KUKA KRL program: EPS_2_25716_MHDR07_A_20250926070400.src

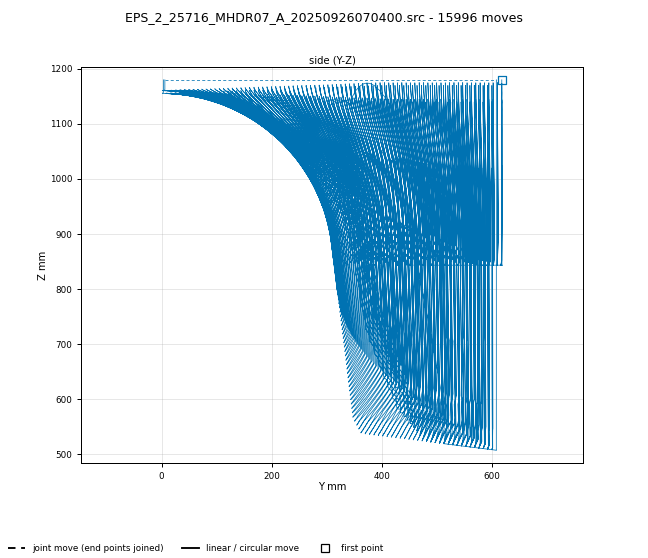
[picture p0: tool path of EPS_2_25716_MHDR07_A_20250926070400.src, 15996 of 15998 moves have a stored position in this frame; points joined in program order, loops and branches not executed]
&ACCESS RVP
&REL 4
&COMMENT QRS 19112012
&PARAM EDITMASK = *
DEF PART()
EXT BAS (BAS_COMMAND :IN,REAL :IN )
INT I
BAS (#INITMOV,0 )

;KUKA QRS Post kuka4.cps  Date:22-06-2017 !

File_ID=2856

QRS_PRE_INIT()

;Init var - Until changes are made in qrs_pre_init
Outlet_Square_prg=0
Inlet_1_Square_prg=0
Inlet_2_Square_prg=0
Inlet_3_Square_prg=0
Inlet_4_Square_prg=0
Inlet_5_Square_prg=0

Outlet_1={X 0.000, Y 400.000, Z 865.000, B 0.000, E1 0.000 }
Inlet_1={X 0.000, Y 425.000, Z 873.500, B 0.000, E1 180.000 }
Inlet_2={X 0.000, Y 495.250, Z 870.500, B 0.000, E1 270.000 }
Outlet_1_type=610
Inlet_1_type=533
Inlet_2_type=299
;QRS#1=Sidecore dimensions
;QRS#2=600-24" Concrete
;QRS#3=525-21" Concrete
;QRS#4=300-12" PVC SDR 35
;QRS#5=
;QRS#6=
;QRS#7=
;QRS#8=
;QRS#9=S306-34L
;QRS#10=S306-32
;QRS#11=16M PSX
;QRS#12=
;QRS#13=
;QRS#14=
;QRS#15=
;QRS#16=1220x127x1524 5'
;QRS#17=EPS Height
;QRS#18=1170
;QRS#19=*
;QRS#20= UPDATED VERSION 22-06-2017
;QRS#21=*
Outlet_Square=0450
Inlet_1_Square=0250
Inlet_2_Square=0150
Inlet_3_Square=0
Inlet_4_Square=0
Inlet_5_Square=0
Mill_Square=1
Outlet_Square_Prg=264
Inlet_1_Square_prg=263
Inlet_2_Square_prg=206

QRS_INIT()

$ADVANCE=5

; T1
PTP {E1 171.027,E2 171.027}
PTP {X 0,Y 617.826,A -85,B 0,C 180,E1 171.027,E2 171.027,E3 0,E4 0,E5 0,E6 0}
QRS_SPEED_INIT()
LIN {X 0,Y 617.826,Z 1180,A -85,B 0,C 180,E1 171.027,E2 171.027,E3 0,E4 0,E5 0,E6 0} C_VEL
LIN {X 0,Y 617.826,Z 845.44,A -85,B 0,C 180,E1 171.027,E2 171.027} C_VEL
LIN {X 0,Y 617.859,Z 843.44,A -85,B 0,C 180,E1 171.213,E2 171.213} C_VEL
LIN {X 0,Y 618.034,Z 843.44,A -85,B 0,C 180,E1 171.886,E2 171.886} C_VEL
LIN {X 0,Y 618.05,Z 843.44,A -85,B 0,C 180,E1 176.532,E2 176.532} C_VEL
LIN {X 0,Y 618.064,Z 843.44,A -85,B 0,C 180,E1 181.155,E2 181.155} C_VEL
LIN {X 0,Y 618.028,Z 843.44,A -85,B 0,C 180,E1 185.786,E2 185.786} C_VEL
LIN {X 0,Y 618.013,Z 843.44,A -85,B 0,C 180,E1 190.456,E2 190.456} C_VEL
LIN {X 0,Y 617.976,Z 843.44,A -85,B 0,C 180,E1 195.197,E2 195.197} C_VEL
LIN {X 0,Y 617.964,Z 843.44,A -85,B 0,C 180,E1 200.048,E2 200.048} C_VEL
LIN {X 0,Y 617.483,Z 843.44,A -85,B 0,C 180,E1 202.547,E2 202.547} C_VEL
LIN {X 0,Y 617.935,Z 843.44,A -85,B 0,C 180,E1 205.055,E2 205.055} C_VEL
LIN {X 0,Y 617.441,Z 843.44,A -85,B 0,C 180,E1 207.658,E2 207.658} C_VEL
LIN {X 0,Y 617.905,Z 843.44,A -85,B 0,C 180,E1 210.277,E2 210.277} C_VEL
LIN {X 0,Y 617.354,Z 843.44,A -85,B 0,C 180,E1 213.025,E2 213.025} C_VEL
LIN {X 0,Y 617.825,Z 843.44,A -85,B 0,C 180,E1 215.797,E2 215.797} C_VEL
LIN {X 0,Y 617.582,Z 843.44,A -85,B 0,C 180,E1 218.101,E2 218.101} C_VEL
LIN {X 0,Y 617.557,Z 843.44,A -85,B 0,C 180,E1 218.721,E2 218.721} C_VEL
LIN {X 0,Y 617.766,Z 843.44,A -85,B 0,C 180,E1 221.733,E2 221.733} C_VEL
LIN {X 0,Y 617.884,Z 843.44,A -85,B 0,C 180,E1 225.1,E2 225.1} C_VEL
LIN {X 0,Y 617.46,Z 843.44,A -85,B 0,C 180,E1 228.307,E2 228.307} C_VEL
LIN {X 0,Y 617.801,Z 843.44,A -85,B 0,C 180,E1 231.297,E2 231.297} C_VEL
LIN {X 0,Y 617.974,Z 843.44,A -85,B 0,C 180,E1 236.343,E2 236.343} C_VEL
LIN {X 0,Y 617.89,Z 843.44,A -85,B 0,C 180,E1 236.673,E2 236.673} C_VEL
LIN {X 0,Y 617.186,Z 843.44,A -85,B 0,C 180,E1 236.798,E2 236.798} C_VEL
LIN {X 0,Y 616.586,Z 843.475,A -85,B 0,C 180,E1 236.859,E2 236.859} C_VEL
LIN {X 0,Y 617.403,Z 850.998,A -85,B 0,C 180,E1 237.011,E2 237.011} C_VEL
LIN {X 0,Y 617.541,Z 885.56,A -85,B 0,C 180,E1 237.498,E2 237.498} C_VEL
LIN {X 0,Y 617.519,Z 896.888,A -85,B 0,C 180,E1 237.684,E2 237.684} C_VEL
LIN {X 0,Y 617.646,Z 911.266,A -85,B 0,C 180,E1 237.997,E2 237.997} C_VEL
LIN {X 0,Y 617.537,Z 922.217,A -85,B 0,C 180,E1 238.279,E2 238.279} C_VEL
LIN {X 0,Y 617.686,Z 929.329,A -85,B 0,C 180,E1 238.492,E2 238.492} C_VEL
LIN {X 0,Y 617.775,Z 942.058,A -85,B 0,C 180,E1 238.905,E2 238.905} C_VEL
LIN {X 0,Y 617.615,Z 958.173,A -85,B 0,C 180,E1 239.505,E2 239.505} C_VEL
LIN {X 0,Y 617.795,Z 971.272,A -85,B 0,C 180,E1 240.077,E2 240.077} C_VEL
LIN {X 0,Y 617.796,Z 985.604,A -85,B 0,C 180,E1 240.772,E2 240.772} C_VEL
LIN {X 0,Y 617.752,Z 997.603,A -85,B 0,C 180,E1 241.411,E2 241.411} C_VEL
LIN {X 0,Y 617.841,Z 1012.189,A -85,B 0,C 180,E1 242.286,E2 242.286} C_VEL
LIN {X 0,Y 617.838,Z 1025.624,A -85,B 0,C 180,E1 243.174,E2 243.174} C_VEL
LIN {X 0,Y 617.827,Z 1037.892,A -85,B 0,C 180,E1 244.06,E2 244.06} C_VEL
LIN {X 0,Y 617.82,Z 1049.111,A -85,B 0,C 180,E1 244.94,E2 244.94} C_VEL
LIN {X 0,Y 617.852,Z 1060.219,A -85,B 0,C 180,E1 245.887,E2 245.887} C_VEL
LIN {X 0,Y 617.902,Z 1071.184,A -85,B 0,C 180,E1 246.902,E2 246.902} C_VEL
LIN {X 0,Y 617.832,Z 1081.53,A -85,B 0,C 180,E1 247.935,E2 247.935} C_VEL
LIN {X 0,Y 617.851,Z 1091.52,A -85,B 0,C 180,E1 249.023,E2 249.023} C_VEL
LIN {X 0,Y 617.958,Z 1100.894,A -85,B 0,C 180,E1 250.135,E2 250.135} C_VEL
LIN {X 0,Y 617.805,Z 1109.459,A -85,B 0,C 180,E1 251.226,E2 251.226} C_VEL
LIN {X 0,Y 617.799,Z 1117.796,A -85,B 0,C 180,E1 252.389,E2 252.389} C_VEL
LIN {X 0,Y 617.999,Z 1125.735,A -85,B 0,C 180,E1 253.612,E2 253.612} C_VEL
LIN {X 0,Y 617.806,Z 1132.883,A -85,B 0,C 180,E1 254.799,E2 254.799} C_VEL
LIN {X 0,Y 617.803,Z 1140.813,A -85,B 0,C 180,E1 256.29,E2 256.29} C_VEL
LIN {X 0,Y 617.952,Z 1146.479,A -85,B 0,C 180,E1 257.48,E2 257.48} C_VEL
LIN {X 0,Y 617.728,Z 1152.733,A -85,B 0,C 180,E1 258.951,E2 258.951} C_VEL
LIN {X 0,Y 617.808,Z 1157.627,A -85,B 0,C 180,E1 260.287,E2 260.287} C_VEL
LIN {X 0,Y 617.981,Z 1160.314,A -85,B 0,C 180,E1 261.14,E2 261.14} C_VEL
LIN {X 0,Y 617.86,Z 1162.559,A -85,B 0,C 180,E1 261.884,E2 261.884} C_VEL
LIN {X 0,Y 617.747,Z 1165.107,A -85,B 0,C 180,E1 262.815,E2 262.815} C_VEL
LIN {X 0,Y 617.832,Z 1168.205,A -85,B 0,C 180,E1 264.212,E2 264.212} C_VEL
LIN {X 0,Y 617.977,Z 1169.802,A -85,B 0,C 180,E1 265.142,E2 265.142} C_VEL
LIN {X 0,Y 617.8,Z 1171.279,A -85,B 0,C 180,E1 266.068,E2 266.068} C_VEL
LIN {X 0,Y 617.755,Z 1172.831,A -85,B 0,C 180,E1 267.456,E2 267.456} C_VEL
LIN {X 0,Y 617.996,Z 1173.642,A -85,B 0,C 180,E1 268.845,E2 268.845} C_VEL
LIN {X 0,Y 617.667,Z 1173.732,A -85,B 0,C 180,E1 271.156,E2 271.156} C_VEL
LIN {X 0,Y 617.779,Z 1173.15,A -85,B 0,C 180,E1 272.081,E2 272.081} C_VEL
LIN {X 0,Y 617.843,Z 1171.818,A -85,B 0,C 180,E1 273.469,E2 273.469} C_VEL
LIN {X 0,Y 617.732,Z 1170.658,A -85,B 0,C 180,E1 274.396,E2 274.396} C_VEL
LIN {X 0,Y 617.804,Z 1168.213,A -85,B 0,C 180,E1 275.788,E2 275.788} C_VEL
LIN {X 0,Y 617.987,Z 1166.125,A -85,B 0,C 180,E1 276.716,E2 276.716} C_VEL
LIN {X 0,Y 617.83,Z 1163.821,A -85,B 0,C 180,E1 277.65,E2 277.65} C_VEL
LIN {X 0,Y 617.779,Z 1160.464,A -85,B 0,C 180,E1 278.831,E2 278.831} C_VEL
LIN {X 0,Y 617.962,Z 1156.403,A -85,B 0,C 180,E1 280.049,E2 280.049} C_VEL
LIN {X 0,Y 617.793,Z 1151.563,A -85,B 0,C 180,E1 281.342,E2 281.342} C_VEL
LIN {X 0,Y 617.737,Z 1146.524,A -85,B 0,C 180,E1 282.524,E2 282.524} C_VEL
LIN {X 0,Y 617.97,Z 1139.3,A -85,B 0,C 180,E1 284.003,E2 284.003} C_VEL
LIN {X 0,Y 617.801,Z 1131.858,A -85,B 0,C 180,E1 285.375,E2 285.375} C_VEL
LIN {X 0,Y 617.792,Z 1124.027,A -85,B 0,C 180,E1 286.666,E2 286.666} C_VEL
LIN {X 0,Y 617.957,Z 1116.024,A -85,B 0,C 180,E1 287.859,E2 287.859} C_VEL
LIN {X 0,Y 617.818,Z 1107.948,A -85,B 0,C 180,E1 288.977,E2 288.977} C_VEL
LIN {X 0,Y 617.839,Z 1098.142,A -85,B 0,C 180,E1 290.206,E2 290.206} C_VEL
LIN {X 0,Y 617.953,Z 1088.763,A -85,B 0,C 180,E1 291.283,E2 291.283} C_VEL
LIN {X 0,Y 617.848,Z 1078.488,A -85,B 0,C 180,E1 292.376,E2 292.376} C_VEL
LIN {X 0,Y 617.845,Z 1068.723,A -85,B 0,C 180,E1 293.335,E2 293.335} C_VEL
LIN {X 0,Y 617.863,Z 1057.185,A -85,B 0,C 180,E1 294.376,E2 294.376} C_VEL
LIN {X 0,Y 617.852,Z 1046.139,A -85,B 0,C 180,E1 295.298,E2 295.298} C_VEL
LIN {X 0,Y 617.837,Z 1033.554,A -85,B 0,C 180,E1 296.261,E2 296.261} C_VEL
LIN {X 0,Y 617.822,Z 1022.09,A -85,B 0,C 180,E1 297.07,E2 297.07} C_VEL
LIN {X 0,Y 617.849,Z 1008.689,A -85,B 0,C 180,E1 297.929,E2 297.929} C_VEL
LIN {X 0,Y 617.812,Z 994.844,A -85,B 0,C 180,E1 298.735,E2 298.735} C_VEL
LIN {X 0,Y 617.727,Z 983.672,A -85,B 0,C 180,E1 299.334,E2 299.334} C_VEL
LIN {X 0,Y 617.802,Z 968.456,A -85,B 0,C 180,E1 300.051,E2 300.051} C_VEL
LIN {X 0,Y 617.675,Z 953.097,A -85,B 0,C 180,E1 300.694,E2 300.694} C_VEL
LIN {X 0,Y 617.671,Z 944.829,A -85,B 0,C 180,E1 300.998,E2 300.998} C_VEL
LIN {X 0,Y 617.767,Z 935.829,A -85,B 0,C 180,E1 301.299,E2 301.299} C_VEL
LIN {X 0,Y 617.783,Z 926.098,A -85,B 0,C 180,E1 301.604,E2 301.604} C_VEL
LIN {X 0,Y 617.523,Z 910.516,A -85,B 0,C 180,E1 302.028,E2 302.028} C_VEL
LIN {X 0,Y 617.755,Z 895.124,A -85,B 0,C 180,E1 302.336,E2 302.336} C_VEL
LIN {X 0,Y 617.696,Z 875.17,A -85,B 0,C 180,E1 302.644,E2 302.644} C_VEL
LIN {X 0,Y 617.35,Z 850.291,A -85,B 0,C 180,E1 303.002,E2 303.002} C_VEL
LIN {X 0,Y 616.629,Z 843.44,A -85,B 0,C 180,E1 303.146,E2 303.146} C_VEL
LIN {X 0,Y 617.119,Z 843.44,A -85,B 0,C 180,E1 303.195,E2 303.195} C_VEL
LIN {X 0,Y 617.816,Z 843.44,A -85,B 0,C 180,E1 303.308,E2 303.308} C_VEL
LIN {X 0,Y 618.037,Z 843.44,A -85,B 0,C 180,E1 303.607,E2 303.607} C_VEL
LIN {X 0,Y 617.768,Z 843.44,A -85,B 0,C 180,E1 305.801,E2 305.801} C_VEL
LIN {X 0,Y 617.724,Z 843.44,A -85,B 0,C 180,E1 308.117,E2 308.117} C_VEL
LIN {X 0,Y 617.813,Z 843.44,A -85,B 0,C 180,E1 311.73,E2 311.73} C_VEL
LIN {X 0,Y 617.416,Z 843.44,A -85,B 0,C 180,E1 315.057,E2 315.057} C_VEL
LIN {X 0,Y 617.813,Z 843.44,A -85,B 0,C 180,E1 318.27,E2 318.27} C_VEL
LIN {X 0,Y 617.717,Z 843.44,A -85,B 0,C 180,E1 321.884,E2 321.884} C_VEL
LIN {X 0,Y 617.729,Z 843.44,A -85,B 0,C 180,E1 324.196,E2 324.196} C_VEL
LIN {X 0,Y 617.802,Z 843.44,A -85,B 0,C 180,E1 325.791,E2 325.791} C_VEL
LIN {X 0,Y 617.831,Z 843.44,A -85,B 0,C 180,E1 327.004,E2 327.004} C_VEL
LIN {X 0,Y 618.061,Z 843.44,A -85,B 0,C 180,E1 331.451,E2 331.451} C_VEL
LIN {X 0,Y 617.532,Z 843.44,A -85,B 0,C 180,E1 335.24,E2 335.24} C_VEL
LIN {X 0,Y 617.711,Z 843.44,A -85,B 0,C 180,E1 337.462,E2 337.462} C_VEL
LIN {X 0,Y 617.977,Z 843.44,A -85,B 0,C 180,E1 342.394,E2 342.394} C_VEL
LIN {X 0,Y 617.279,Z 843.44,A -85,B 0,C 180,E1 342.777,E2 342.777} C_VEL
LIN {X 0,Y 616.404,Z 843.44,A -85,B 0,C 180,E1 342.867,E2 342.867} C_VEL
LIN {X 0,Y 617.46,Z 848.376,A -85,B 0,C 180,E1 342.958,E2 342.958} C_VEL
LIN {X 0,Y 617.866,Z 852.602,A -85,B 0,C 180,E1 343.02,E2 343.02} C_VEL
LIN {X 0,Y 617.94,Z 873.653,A -85,B 0,C 180,E1 343.286,E2 343.286} C_VEL
LIN {X 0,Y 617.951,Z 884.015,A -85,B 0,C 180,E1 343.474,E2 343.474} C_VEL
LIN {X 0,Y 617.935,Z 894.426,A -85,B 0,C 180,E1 343.73,E2 343.73} C_VEL
LIN {X 0,Y 618.005,Z 903.309,A -85,B 0,C 180,E1 344,E2 344} C_VEL
LIN {X 0,Y 617.986,Z 911.677,A -85,B 0,C 180,E1 344.297,E2 344.297} C_VEL
LIN {X 0,Y 617.988,Z 918.429,A -85,B 0,C 180,E1 344.571,E2 344.571} C_VEL
LIN {X 0,Y 618.018,Z 926.731,A -85,B 0,C 180,E1 344.953,E2 344.953} C_VEL
LIN {X 0,Y 618.01,Z 935.331,A -85,B 0,C 180,E1 345.401,E2 345.401} C_VEL
LIN {X 0,Y 617.98,Z 945.261,A -85,B 0,C 180,E1 345.997,E2 345.997} C_VEL
LIN {X 0,Y 617.998,Z 952.881,A -85,B 0,C 180,E1 346.518,E2 346.518} C_VEL
LIN {X 0,Y 618.001,Z 959.746,A -85,B 0,C 180,E1 347.037,E2 347.037} C_VEL
LIN {X 0,Y 617.986,Z 966.834,A -85,B 0,C 180,E1 347.629,E2 347.629} C_VEL
LIN {X 0,Y 617.989,Z 974.718,A -85,B 0,C 180,E1 348.367,E2 348.367} C_VEL
LIN {X 0,Y 617.99,Z 980.34,A -85,B 0,C 180,E1 348.956,E2 348.956} C_VEL
LIN {X 0,Y 618.005,Z 985.465,A -85,B 0,C 180,E1 349.544,E2 349.544} C_VEL
LIN {X 0,Y 617.972,Z 991.481,A -85,B 0,C 180,E1 350.309,E2 350.309} C_VEL
LIN {X 0,Y 617.952,Z 996.842,A -85,B 0,C 180,E1 351.072,E2 351.072} C_VEL
LIN {X 0,Y 617.99,Z 1001.905,A -85,B 0,C 180,E1 351.886,E2 351.886} C_VEL
LIN {X 0,Y 617.944,Z 1006.92,A -85,B 0,C 180,E1 352.818,E2 352.818} C_VEL
LIN {X 0,Y 617.915,Z 1010.212,A -85,B 0,C 180,E1 353.516,E2 353.516} C_VEL
LIN {X 0,Y 617.956,Z 1013.094,A -85,B 0,C 180,E1 354.213,E2 354.213} C_VEL
LIN {X 0,Y 617.988,Z 1014.821,A -85,B 0,C 180,E1 354.678,E2 354.678} C_VEL
LIN {X 0,Y 617.913,Z 1017.797,A -85,B 0,C 180,E1 355.605,E2 355.605} C_VEL
LIN {X 0,Y 617.894,Z 1020.135,A -85,B 0,C 180,E1 356.531,E2 356.531} C_VEL
LIN {X 0,Y 617.975,Z 1021.885,A -85,B 0,C 180,E1 357.457,E2 357.457} C_VEL
LIN {X 0,Y 617.978,Z 1022.566,A -85,B 0,C 180,E1 357.92,E2 357.92} C_VEL
LIN {X 0,Y 617.893,Z 1023.509,A -85,B 0,C 180,E1 358.844,E2 358.844} C_VEL
LIN {X 0,Y 617.884,Z 1023.799,A -85,B 0,C 180,E1 359.307,E2 359.307} C_VEL
LIN {X 0,Y 617.958,Z 1023.865,A -85,B 0,C 180,E1 360.231,E2 360.231} C_VEL
LIN {X 0,Y 617.93,Z 1023.435,A -85,B 0,C 180,E1 361.156,E2 361.156} C_VEL
LIN {X 0,Y 617.886,Z 1023.032,A -85,B 0,C 180,E1 361.618,E2 361.618} C_VEL
LIN {X 0,Y 617.897,Z 1021.756,A -85,B 0,C 180,E1 362.543,E2 362.543} C_VEL
LIN {X 0,Y 617.989,Z 1019.915,A -85,B 0,C 180,E1 363.468,E2 363.468} C_VEL
LIN {X 0,Y 617.905,Z 1017.555,A -85,B 0,C 180,E1 364.395,E2 364.395} C_VEL
LIN {X 0,Y 617.893,Z 1014.509,A -85,B 0,C 180,E1 365.323,E2 365.323} C_VEL
LIN {X 0,Y 617.929,Z 1012.766,A -85,B 0,C 180,E1 365.787,E2 365.787} C_VEL
LIN {X 0,Y 617.981,Z 1008.74,A -85,B 0,C 180,E1 366.716,E2 366.716} C_VEL
LIN {X 0,Y 617.924,Z 1004.006,A -85,B 0,C 180,E1 367.649,E2 367.649} C_VEL
LIN {X 0,Y 617.961,Z 998.442,A -85,B 0,C 180,E1 368.595,E2 368.595} C_VEL
LIN {X 0,Y 618.003,Z 993.303,A -85,B 0,C 180,E1 369.355,E2 369.355} C_VEL
LIN {X 0,Y 617.953,Z 987.738,A -85,B 0,C 180,E1 370.089,E2 370.089} C_VEL
LIN {X 0,Y 617.968,Z 982.163,A -85,B 0,C 180,E1 370.75,E2 370.75} C_VEL
LIN {X 0,Y 618.001,Z 975.273,A -85,B 0,C 180,E1 371.485,E2 371.485} C_VEL
LIN {X 0,Y 617.99,Z 967.501,A -85,B 0,C 180,E1 372.223,E2 372.223} C_VEL
LIN {X 0,Y 617.991,Z 960.481,A -85,B 0,C 180,E1 372.815,E2 372.815} C_VEL
LIN {X 0,Y 618.01,Z 953.686,A -85,B 0,C 180,E1 373.334,E2 373.334} C_VEL
LIN {X 0,Y 618.026,Z 946.145,A -85,B 0,C 180,E1 373.853,E2 373.853} C_VEL
LIN {X 0,Y 618.015,Z 936.423,A -85,B 0,C 180,E1 374.449,E2 374.449} C_VEL
LIN {X 0,Y 617.982,Z 927.966,A -85,B 0,C 180,E1 374.898,E2 374.898} C_VEL
LIN {X 0,Y 618.015,Z 919.027,A -85,B 0,C 180,E1 375.312,E2 375.312} C_VEL
LIN {X 0,Y 618.031,Z 910.408,A -85,B 0,C 180,E1 375.66,E2 375.66} C_VEL
LIN {X 0,Y 617.966,Z 901.85,A -85,B 0,C 180,E1 375.959,E2 375.959} C_VEL
LIN {X 0,Y 618.01,Z 891.38,A -85,B 0,C 180,E1 376.262,E2 376.262} C_VEL
LIN {X 0,Y 617.964,Z 880.659,A -85,B 0,C 180,E1 376.501,E2 376.501} C_VEL
LIN {X 0,Y 617.886,Z 871.697,A -85,B 0,C 180,E1 376.653,E2 376.653} C_VEL
LIN {X 0,Y 617.825,Z 844.104,A -85,B 0,C 180,E1 376.992,E2 376.992} C_VEL
LIN {X 0,Y 617.73,Z 843.44,A -85,B 0,C 180,E1 377.012,E2 377.012} C_VEL
LIN {X 0,Y 618.008,Z 843.44,A -85,B 0,C 180,E1 377.344,E2 377.344} C_VEL
LIN {X 0,Y 617.906,Z 843.44,A -85,B 0,C 180,E1 382.53,E2 382.53} C_VEL
LIN {X 0,Y 617.419,Z 843.44,A -85,B 0,C 180,E1 385.077,E2 385.077} C_VEL
LIN {X 0,Y 617.864,Z 843.44,A -85,B 0,C 180,E1 387.637,E2 387.637} C_VEL
LIN {X 0,Y 617.41,Z 843.44,A -85,B 0,C 180,E1 390.304,E2 390.304} C_VEL
LIN {X 0,Y 617.944,Z 843.44,A -85,B 0,C 180,E1 392.989,E2 392.989} C_VEL
LIN {X 0,Y 617.692,Z 843.44,A -85,B 0,C 180,E1 395.806,E2 395.806} C_VEL
LIN {X 0,Y 617.698,Z 843.44,A -85,B 0,C 180,E1 398.114,E2 398.114} C_VEL
LIN {X 0,Y 617.763,Z 843.44,A -85,B 0,C 180,E1 401.734,E2 401.734} C_VEL
LIN {X 0,Y 617.403,Z 843.44,A -85,B 0,C 180,E1 405.055,E2 405.055} C_VEL
LIN {X 0,Y 617.813,Z 843.44,A -85,B 0,C 180,E1 408.27,E2 408.27} C_VEL
LIN {X 0,Y 617.726,Z 843.44,A -85,B 0,C 180,E1 411.882,E2 411.882} C_VEL
LIN {X 0,Y 617.761,Z 843.44,A -85,B 0,C 180,E1 414.198,E2 414.198} C_VEL
LIN {X 0,Y 617.859,Z 843.44,A -85,B 0,C 180,E1 415.783,E2 415.783} C_VEL
LIN {X 0,Y 617.919,Z 843.44,A -85,B 0,C 180,E1 417.01,E2 417.01} C_VEL
LIN {X 0,Y 618.055,Z 843.44,A -85,B 0,C 180,E1 420.692,E2 420.692} C_VEL
LIN {X 0,Y 616.955,Z 843.44,A -85,B 0,C 180,E1 420.924,E2 420.924} C_VEL
LIN {X 0,Y 617.601,Z 885.711,A -85,B 0,C 180,E1 421.513,E2 421.513} C_VEL
LIN {X 0,Y 617.776,Z 900.46,A -85,B 0,C 180,E1 421.761,E2 421.761} C_VEL
LIN {X 0,Y 617.725,Z 913.777,A -85,B 0,C 180,E1 422.041,E2 422.041} C_VEL
LIN {X 0,Y 617.739,Z 922.091,A -85,B 0,C 180,E1 422.252,E2 422.252} C_VEL
LIN {X 0,Y 617.888,Z 937.972,A -85,B 0,C 180,E1 422.73,E2 422.73} C_VEL
LIN {X 0,Y 617.81,Z 952.541,A -85,B 0,C 180,E1 423.253,E2 423.253} C_VEL
LIN {X 0,Y 617.771,Z 960.477,A -85,B 0,C 180,E1 423.575,E2 423.575} C_VEL
LIN {X 0,Y 617.905,Z 974.757,A -85,B 0,C 180,E1 424.224,E2 424.224} C_VEL
LIN {X 0,Y 617.888,Z 988.689,A -85,B 0,C 180,E1 424.943,E2 424.943} C_VEL
LIN {X 0,Y 617.879,Z 1000.176,A -85,B 0,C 180,E1 425.605,E2 425.605} C_VEL
LIN {X 0,Y 617.914,Z 1012.714,A -85,B 0,C 180,E1 426.41,E2 426.41} C_VEL
LIN {X 0,Y 617.927,Z 1023.539,A -85,B 0,C 180,E1 427.173,E2 427.173} C_VEL
LIN {X 0,Y 617.917,Z 1033.547,A -85,B 0,C 180,E1 427.938,E2 427.938} C_VEL
LIN {X 0,Y 617.883,Z 1044.646,A -85,B 0,C 180,E1 428.869,E2 428.869} C_VEL
LIN {X 0,Y 617.917,Z 1053.151,A -85,B 0,C 180,E1 429.643,E2 429.643} C_VEL
LIN {X 0,Y 617.951,Z 1061.756,A -85,B 0,C 180,E1 430.489,E2 430.489} C_VEL
LIN {X 0,Y 617.881,Z 1070.527,A -85,B 0,C 180,E1 431.422,E2 431.422} C_VEL
LIN {X 0,Y 617.893,Z 1078.874,A -85,B 0,C 180,E1 432.391,E2 432.391} C_VEL
LIN {X 0,Y 617.963,Z 1087.602,A -85,B 0,C 180,E1 433.508,E2 433.508} C_VEL
LIN {X 0,Y 617.843,Z 1095.506,A -85,B 0,C 180,E1 434.61,E2 434.61} C_VEL
LIN {X 0,Y 617.862,Z 1100.731,A -85,B 0,C 180,E1 435.398,E2 435.398} C_VEL
LIN {X 0,Y 617.952,Z 1107.875,A -85,B 0,C 180,E1 436.591,E2 436.591} C_VEL
LIN {X 0,Y 617.775,Z 1114.283,A -85,B 0,C 180,E1 437.772,E2 437.772} C_VEL
LIN {X 0,Y 617.807,Z 1119.937,A -85,B 0,C 180,E1 438.953,E2 438.953} C_VEL
LIN {X 0,Y 617.959,Z 1124.156,A -85,B 0,C 180,E1 439.949,E2 439.949} C_VEL
LIN {X 0,Y 617.802,Z 1129.113,A -85,B 0,C 180,E1 441.247,E2 441.247} C_VEL
LIN {X 0,Y 617.807,Z 1132.662,A -85,B 0,C 180,E1 442.35,E2 442.35} C_VEL
LIN {X 0,Y 617.966,Z 1136.451,A -85,B 0,C 180,E1 443.749,E2 443.749} C_VEL
LIN {X 0,Y 617.739,Z 1139.478,A -85,B 0,C 180,E1 445.14,E2 445.14} C_VEL
LIN {X 0,Y 617.821,Z 1141.652,A -85,B 0,C 180,E1 446.531,E2 446.531} C_VEL
LIN {X 0,Y 617.873,Z 1143.084,A -85,B 0,C 180,E1 447.92,E2 447.92} C_VEL
LIN {X 0,Y 617.751,Z 1143.724,A -85,B 0,C 180,E1 448.844,E2 448.844} C_VEL
LIN {X 0,Y 617.981,Z 1143.64,A -85,B 0,C 180,E1 451.155,E2 451.155} C_VEL
LIN {X 0,Y 617.795,Z 1142.66,A -85,B 0,C 180,E1 452.543,E2 452.543} C_VEL
LIN {X 0,Y 617.867,Z 1140.852,A -85,B 0,C 180,E1 453.932,E2 453.932} C_VEL
LIN {X 0,Y 617.954,Z 1139.273,A -85,B 0,C 180,E1 454.858,E2 454.858} C_VEL
LIN {X 0,Y 617.735,Z 1136.276,A -85,B 0,C 180,E1 456.254,E2 456.254} C_VEL
LIN {X 0,Y 617.833,Z 1132.365,A -85,B 0,C 180,E1 457.65,E2 457.65} C_VEL
LIN {X 0,Y 617.997,Z 1129.526,A -85,B 0,C 180,E1 458.521,E2 458.521} C_VEL
LIN {X 0,Y 617.81,Z 1125.257,A -85,B 0,C 180,E1 459.694,E2 459.694} C_VEL
LIN {X 0,Y 617.829,Z 1119.54,A -85,B 0,C 180,E1 461.047,E2 461.047} C_VEL
LIN {X 0,Y 617.965,Z 1113.799,A -85,B 0,C 180,E1 462.224,E2 462.224} C_VEL
LIN {X 0,Y 617.825,Z 1107.383,A -85,B 0,C 180,E1 463.412,E2 463.412} C_VEL
LIN {X 0,Y 617.883,Z 1100.129,A -85,B 0,C 180,E1 464.602,E2 464.602} C_VEL
LIN {X 0,Y 617.971,Z 1093.663,A -85,B 0,C 180,E1 465.57,E2 465.57} C_VEL
LIN {X 0,Y 617.855,Z 1084.805,A -85,B 0,C 180,E1 466.775,E2 466.775} C_VEL
LIN {X 0,Y 617.908,Z 1077.009,A -85,B 0,C 180,E1 467.74,E2 467.74} C_VEL
LIN {X 0,Y 617.968,Z 1068.894,A -85,B 0,C 180,E1 468.664,E2 468.664} C_VEL
LIN {X 0,Y 617.888,Z 1058.94,A -85,B 0,C 180,E1 469.704,E2 469.704} C_VEL
LIN {X 0,Y 617.909,Z 1050.523,A -85,B 0,C 180,E1 470.512,E2 470.512} C_VEL
LIN {X 0,Y 617.926,Z 1039.982,A -85,B 0,C 180,E1 471.439,E2 471.439} C_VEL
LIN {X 0,Y 617.908,Z 1030.394,A -85,B 0,C 180,E1 472.218,E2 472.218} C_VEL
LIN {X 0,Y 617.903,Z 1020.403,A -85,B 0,C 180,E1 472.966,E2 472.966} C_VEL
LIN {X 0,Y 617.9,Z 1008.891,A -85,B 0,C 180,E1 473.753,E2 473.753} C_VEL
LIN {X 0,Y 617.897,Z 998.001,A -85,B 0,C 180,E1 474.433,E2 474.433} C_VEL
LIN {X 0,Y 617.868,Z 985.501,A -85,B 0,C 180,E1 475.138,E2 475.138} C_VEL
LIN {X 0,Y 617.805,Z 974.544,A -85,B 0,C 180,E1 475.7,E2 475.7} C_VEL
LIN {X 0,Y 617.902,Z 962.228,A -85,B 0,C 180,E1 476.258,E2 476.258} C_VEL
LIN {X 0,Y 617.838,Z 948.02,A -85,B 0,C 180,E1 476.826,E2 476.826} C_VEL
LIN {X 0,Y 617.71,Z 936.079,A -85,B 0,C 180,E1 477.248,E2 477.248} C_VEL
LIN {X 0,Y 617.845,Z 922.678,A -85,B 0,C 180,E1 477.638,E2 477.638} C_VEL
LIN {X 0,Y 617.775,Z 908.541,A -85,B 0,C 180,E1 477.985,E2 477.985} C_VEL
LIN {X 0,Y 617.68,Z 898.255,A -85,B 0,C 180,E1 478.198,E2 478.198} C_VEL
LIN {X 0,Y 617.702,Z 879.224,A -85,B 0,C 180,E1 478.477,E2 478.477} C_VEL
LIN {X 0,Y 617.587,Z 857.783,A -85,B 0,C 180,E1 478.762,E2 478.762} C_VEL
LIN {X 0,Y 617.384,Z 852.419,A -85,B 0,C 180,E1 478.842,E2 478.842} C_VEL
LIN {X 0,Y 616.533,Z 844.921,A -85,B 0,C 180,E1 478.983,E2 478.983} C_VEL
LIN {X 0,Y 616.607,Z 843.44,A -85,B 0,C 180,E1 479.035,E2 479.035} C_VEL
LIN {X 0,Y 616.994,Z 843.44,A -85,B 0,C 180,E1 479.071,E2 479.071} C_VEL
LIN {X 0,Y 617.992,Z 843.44,A -85,B 0,C 180,E1 479.266,E2 479.266} C_VEL
LIN {X 0,Y 618.022,Z 843.44,A -85,B 0,C 180,E1 480.27,E2 480.27} C_VEL
LIN {X 0,Y 617.371,Z 843.44,A -85,B 0,C 180,E1 484.15,E2 484.15} C_VEL
LIN {X 0,Y 617.838,Z 843.44,A -85,B 0,C 180,E1 485.797,E2 485.797} C_VEL
LIN {X 0,Y 617.927,Z 843.44,A -85,B 0,C 180,E1 488.694,E2 488.694} C_VEL
LIN {X 0,Y 617.445,Z 843.44,A -85,B 0,C 180,E1 491.76,E2 491.76} C_VEL
LIN {X 0,Y 617.887,Z 843.44,A -85,B 0,C 180,E1 494.9,E2 494.9} C_VEL
LIN {X 0,Y 617.774,Z 843.44,A -85,B 0,C 180,E1 498.274,E2 498.274} C_VEL
LIN {X 0,Y 617.55,Z 843.44,A -85,B 0,C 180,E1 501.278,E2 501.278} C_VEL
LIN {X 0,Y 617.814,Z 843.44,A -85,B 0,C 180,E1 504.202,E2 504.202} C_VEL
LIN {X 0,Y 617.349,Z 843.44,A -85,B 0,C 180,E1 506.975,E2 506.975} C_VEL
LIN {X 0,Y 617.905,Z 843.44,A -85,B 0,C 180,E1 509.723,E2 509.723} C_VEL
LIN {X 0,Y 617.442,Z 843.44,A -85,B 0,C 180,E1 512.342,E2 512.342} C_VEL
LIN {X 0,Y 617.936,Z 843.44,A -85,B 0,C 180,E1 514.945,E2 514.945} C_VEL
LIN {X 0,Y 617.486,Z 843.44,A -85,B 0,C 180,E1 517.453,E2 517.453} C_VEL
LIN {X 0,Y 617.991,Z 843.44,A -85,B 0,C 180,E1 519.953,E2 519.953} C_VEL
LIN {X 0,Y 617.756,Z 843.44,A -85,B 0,C 180,E1 522.387,E2 522.387} C_VEL
LIN {X 0,Y 617.825,Z 843.44,A -85,B 0,C 180,E1 524.799,E2 524.799} C_VEL
LIN {X 0,Y 617.986,Z 843.44,A -85,B 0,C 180,E1 527.185,E2 527.185} C_VEL
LIN {X 0,Y 617.859,Z 843.44,A -85,B 0,C 180,E1 531.213,E2 531.213} C_VEL
LIN {X 0,Y 615.328,Z 843.44,A -85,B 0,C 180,E1 532.409,E2 532.409} C_VEL
LIN {X 0,Y 609.74,Z 843.44,A -85,B 0,C 180,E1 534.196,E2 534.196} C_VEL
LIN {X 0,Y 609.651,Z 843.44,A -85,B 0,C 180,E1 534.403,E2 534.403} C_VEL
LIN {X 0,Y 609.661,Z 843.44,A -85,B 0,C 180,E1 538.578,E2 538.578} C_VEL
LIN {X 0,Y 609.695,Z 843.44,A -85,B 0,C 180,E1 542.847,E2 542.847} C_VEL
LIN {X 0,Y 609.729,Z 843.44,A -85,B 0,C 180,E1 547.132,E2 547.132} C_VEL
LIN {X 0,Y 609.778,Z 843.44,A -85,B 0,C 180,E1 551.457,E2 551.457} C_VEL
LIN {X 0,Y 609.814,Z 843.44,A -85,B 0,C 180,E1 555.849,E2 555.849} C_VEL
LIN {X 0,Y 609.973,Z 843.44,A -85,B 0,C 180,E1 560.334,E2 560.334} C_VEL
LIN {X 0,Y 610.019,Z 843.44,A -85,B 0,C 180,E1 564.956,E2 564.956} C_VEL
LIN {X 0,Y 609.824,Z 843.44,A -85,B 0,C 180,E1 569.771,E2 569.771} C_VEL
LIN {X 0,Y 609.762,Z 843.44,A -85,B 0,C 180,E1 576.576,E2 576.576} C_VEL
LIN {X 0,Y 609.775,Z 843.44,A -85,B 0,C 180,E1 582.095,E2 582.095} C_VEL
LIN {X 0,Y 609.525,Z 843.44,A -85,B 0,C 180,E1 587.879,E2 587.879} C_VEL
LIN {X 0,Y 609.494,Z 843.44,A -85,B 0,C 180,E1 592.643,E2 592.643} C_VEL
LIN {X 0,Y 610.005,Z 843.44,A -85,B 0,C 180,E1 596.454,E2 596.454} C_VEL
LIN {X 0,Y 610.914,Z 911.028,A -85,B 0,C 180,E1 597.596,E2 597.596} C_VEL
LIN {X 0,Y 610.806,Z 953.607,A -85,B 0,C 180,E1 598.942,E2 598.942} C_VEL
LIN {X 0,Y 610.644,Z 994.599,A -85,B 0,C 180,E1 600.882,E2 600.882} C_VEL
LIN {X 0,Y 610.514,Z 1032.281,A -85,B 0,C 180,E1 603.307,E2 603.307} C_VEL
LIN {X 0,Y 610.326,Z 1066.547,A -85,B 0,C 180,E1 606.159,E2 606.159} C_VEL
LIN {X 0,Y 610.191,Z 1096.181,A -85,B 0,C 180,E1 609.293,E2 609.293} C_VEL
LIN {X 0,Y 610.072,Z 1121.358,A -85,B 0,C 180,E1 612.674,E2 612.674} C_VEL
LIN {X 0,Y 610.012,Z 1142.477,A -85,B 0,C 180,E1 616.362,E2 616.362} C_VEL
LIN {X 0,Y 609.953,Z 1157.781,A -85,B 0,C 180,E1 619.994,E2 619.994} C_VEL
LIN {X 0,Y 609.942,Z 1167.915,A -85,B 0,C 180,E1 623.586,E2 623.586} C_VEL
LIN {X 0,Y 609.916,Z 1173.628,A -85,B 0,C 180,E1 627.155,E2 627.155} C_VEL
LIN {X 0,Y 609.939,Z 1175,A -85,B 0,C 180,E1 630.001,E2 630.001} C_VEL
LIN {X 0,Y 609.985,Z 1173.626,A -85,B 0,C 180,E1 632.846,E2 632.846} C_VEL
LIN {X 0,Y 610.092,Z 1166.329,A -85,B 0,C 180,E1 637.129,E2 637.129} C_VEL
LIN {X 0,Y 609.998,Z 1153.73,A -85,B 0,C 180,E1 641.092,E2 641.092} C_VEL
LIN {X 0,Y 610.028,Z 1135.009,A -85,B 0,C 180,E1 645.071,E2 645.071} C_VEL
LIN {X 0,Y 610.137,Z 1112.342,A -85,B 0,C 180,E1 648.634,E2 648.634} C_VEL
LIN {X 0,Y 610.266,Z 1084.394,A -85,B 0,C 180,E1 652.042,E2 652.042} C_VEL
LIN {X 0,Y 610.39,Z 1051.996,A -85,B 0,C 180,E1 655.139,E2 655.139} C_VEL
LIN {X 0,Y 610.589,Z 1017.429,A -85,B 0,C 180,E1 657.725,E2 657.725} C_VEL
LIN {X 0,Y 610.729,Z 979.431,A -85,B 0,C 180,E1 659.91,E2 659.91} C_VEL
LIN {X 0,Y 610.944,Z 939.579,A -85,B 0,C 180,E1 661.569,E2 661.569} C_VEL
LIN {X 0,Y 611.009,Z 900.073,A -85,B 0,C 180,E1 662.635,E2 662.635} C_VEL
LIN {X 0,Y 610.017,Z 843.44,A -85,B 0,C 180,E1 663.547,E2 663.547} C_VEL
LIN {X 0,Y 609.756,Z 843.44,A -85,B 0,C 180,E1 668.375,E2 668.375} C_VEL
LIN {X 0,Y 609.761,Z 843.44,A -85,B 0,C 180,E1 672.103,E2 672.103} C_VEL
LIN {X 0,Y 609.856,Z 843.44,A -85,B 0,C 180,E1 678.146,E2 678.146} C_VEL
LIN {X 0,Y 609.735,Z 843.44,A -85,B 0,C 180,E1 683.422,E2 683.422} C_VEL
LIN {X 0,Y 609.757,Z 843.44,A -85,B 0,C 180,E1 687.596,E2 687.596} C_VEL
LIN {X 0,Y 609.98,Z 843.44,A -85,B 0,C 180,E1 691.863,E2 691.863} C_VEL
LIN {X 0,Y 609.587,Z 843.44,A -85,B 0,C 180,E1 698.127,E2 698.127} C_VEL
LIN {X 0,Y 609.583,Z 843.44,A -85,B 0,C 180,E1 701.163,E2 701.163} C_VEL
LIN {X 0,Y 608.887,Z 843.44,A -85,B 0,C 180,E1 702.64,E2 702.64} C_VEL
LIN {X 0,Y 610.388,Z 865.576,A -85,B 0,C 180,E1 702.963,E2 702.963} C_VEL
LIN {X 0,Y 610.381,Z 897.548,A -85,B 0,C 180,E1 703.612,E2 703.612} C_VEL
LIN {X 0,Y 610.359,Z 927.083,A -85,B 0,C 180,E1 704.773,E2 704.773} C_VEL
LIN {X 0,Y 610.27,Z 954.696,A -85,B 0,C 180,E1 706.459,E2 706.459} C_VEL
LIN {X 0,Y 610.228,Z 978.366,A -85,B 0,C 180,E1 708.551,E2 708.551} C_VEL
LIN {X 0,Y 610.157,Z 998.305,A -85,B 0,C 180,E1 711.078,E2 711.078} C_VEL
LIN {X 0,Y 610.128,Z 1011.715,A -85,B 0,C 180,E1 713.588,E2 713.588} C_VEL
LIN {X 0,Y 610.081,Z 1021.032,A -85,B 0,C 180,E1 716.443,E2 716.443} C_VEL
LIN {X 0,Y 610.084,Z 1024.382,A -85,B 0,C 180,E1 718.577,E2 718.577} C_VEL
LIN {X 0,Y 610.079,Z 1024.317,A -85,B 0,C 180,E1 721.421,E2 721.421} C_VEL
LIN {X 0,Y 610.112,Z 1019.005,A -85,B 0,C 180,E1 724.269,E2 724.269} C_VEL
LIN {X 0,Y 610.145,Z 1008,A -85,B 0,C 180,E1 727.126,E2 727.126} C_VEL
LIN {X 0,Y 610.2,Z 991.371,A -85,B 0,C 180,E1 729.82,E2 729.82} C_VEL
LIN {X 0,Y 610.229,Z 970.136,A -85,B 0,C 180,E1 732.173,E2 732.173} C_VEL
LIN {X 0,Y 610.342,Z 944.151,A -85,B 0,C 180,E1 734.178,E2 734.178} C_VEL
LIN {X 0,Y 610.412,Z 914.929,A -85,B 0,C 180,E1 735.689,E2 735.689} C_VEL
LIN {X 0,Y 610.444,Z 885.213,A -85,B 0,C 180,E1 736.617,E2 736.617} C_VEL
LIN {X 0,Y 609.99,Z 843.44,A -85,B 0,C 180,E1 737.233,E2 737.233} C_VEL
LIN {X 0,Y 609.718,Z 843.44,A -85,B 0,C 180,E1 743.408,E2 743.408} C_VEL
LIN {X 0,Y 609.783,Z 843.44,A -85,B 0,C 180,E1 748.145,E2 748.145} C_VEL
LIN {X 0,Y 610.005,Z 843.44,A -85,B 0,C 180,E1 753.093,E2 753.093} C_VEL
LIN {X 0,Y 609.734,Z 843.44,A -85,B 0,C 180,E1 758.369,E2 758.369} C_VEL
LIN {X 0,Y 609.742,Z 843.44,A -85,B 0,C 180,E1 762.096,E2 762.096} C_VEL
LIN {X 0,Y 609.865,Z 843.44,A -85,B 0,C 180,E1 768.135,E2 768.135} C_VEL
LIN {X 0,Y 609.757,Z 843.44,A -85,B 0,C 180,E1 773.418,E2 773.418} C_VEL
LIN {X 0,Y 609.793,Z 843.44,A -85,B 0,C 180,E1 778.571,E2 778.571} C_VEL
LIN {X 0,Y 610.098,Z 843.44,A -85,B 0,C 180,E1 780.547,E2 780.547} C_VEL
LIN {X 0,Y 610.772,Z 911.897,A -85,B 0,C 180,E1 781.647,E2 781.647} C_VEL
LIN {X 0,Y 610.672,Z 952.862,A -85,B 0,C 180,E1 782.929,E2 782.929} C_VEL
LIN {X 0,Y 610.547,Z 991.246,A -85,B 0,C 180,E1 784.77,E2 784.77} C_VEL
LIN {X 0,Y 610.417,Z 1026.435,A -85,B 0,C 180,E1 787.099,E2 787.099} C_VEL
LIN {X 0,Y 610.268,Z 1057.42,A -85,B 0,C 180,E1 789.797,E2 789.797} C_VEL
LIN {X 0,Y 610.184,Z 1084.542,A -85,B 0,C 180,E1 792.862,E2 792.862} C_VEL
LIN {X 0,Y 610.154,Z 1108.014,A -85,B 0,C 180,E1 796.364,E2 796.364} C_VEL
LIN {X 0,Y 610.133,Z 1125.586,A -85,B 0,C 180,E1 799.995,E2 799.995} C_VEL
LIN {X 0,Y 610.136,Z 1137.153,A -85,B 0,C 180,E1 803.587,E2 803.587} C_VEL
LIN {X 0,Y 609.984,Z 1143.447,A -85,B 0,C 180,E1 807.154,E2 807.154} C_VEL
LIN {X 0,Y 609.957,Z 1144.996,A -85,B 0,C 180,E1 809.999,E2 809.999} C_VEL
LIN {X 0,Y 609.953,Z 1143.341,A -85,B 0,C 180,E1 812.845,E2 812.845} C_VEL
LIN {X 0,Y 609.9,Z 1136.915,A -85,B 0,C 180,E1 816.414,E2 816.414} C_VEL
LIN {X 0,Y 610.004,Z 1126.607,A -85,B 0,C 180,E1 819.645,E2 819.645} C_VEL
LIN {X 0,Y 610.044,Z 1109.546,A -85,B 0,C 180,E1 823.272,E2 823.272} C_VEL
LIN {X 0,Y 610.124,Z 1086.765,A -85,B 0,C 180,E1 826.767,E2 826.767} C_VEL
LIN {X 0,Y 610.243,Z 1059.166,A -85,B 0,C 180,E1 829.942,E2 829.942} C_VEL
LIN {X 0,Y 610.393,Z 1027.787,A -85,B 0,C 180,E1 832.708,E2 832.708} C_VEL
LIN {X 0,Y 610.551,Z 993.094,A -85,B 0,C 180,E1 835.032,E2 835.032} C_VEL
LIN {X 0,Y 610.716,Z 956.661,A -85,B 0,C 180,E1 836.822,E2 836.822} C_VEL
LIN {X 0,Y 610.824,Z 922.007,A -85,B 0,C 180,E1 838.002,E2 838.002} C_VEL
LIN {X 0,Y 610.802,Z 884.946,A -85,B 0,C 180,E1 838.754,E2 838.754} C_VEL
LIN {X 0,Y 609.718,Z 843.44,A -85,B 0,C 180,E1 839.393,E2 839.393} C_VEL
LIN {X 0,Y 609.661,Z 843.44,A -85,B 0,C 180,E1 844.969,E2 844.969} C_VEL
LIN {X 0,Y 609.691,Z 843.44,A -85,B 0,C 180,E1 849.668,E2 849.668} C_VEL
LIN {X 0,Y 609.733,Z 843.44,A -85,B 0,C 180,E1 855.956,E2 855.956} C_VEL
LIN {X 0,Y 609.539,Z 843.44,A -85,B 0,C 180,E1 860.358,E2 860.358} C_VEL
LIN {X 0,Y 609.603,Z 843.44,A -85,B 0,C 180,E1 865.167,E2 865.167} C_VEL
LIN {X 0,Y 609.779,Z 843.44,A -85,B 0,C 180,E1 870.351,E2 870.351} C_VEL
LIN {X 0,Y 610.02,Z 843.44,A -85,B 0,C 180,E1 875.046,E2 875.046} C_VEL
LIN {X 0,Y 609.863,Z 843.44,A -85,B 0,C 180,E1 881.173,E2 881.173} C_VEL
LIN {X 0,Y 610.076,Z 843.44,A -85,B 0,C 180,E1 887.095,E2 887.095} C_VEL
LIN {X 0,Y 609.816,Z 843.44,A -85,B 0,C 180,E1 892.87,E2 892.87} C_VEL
LIN {X 0,Y 609.651,Z 843.44,A -85,B 0,C 180,E1 894.403,E2 894.403} C_VEL
LIN {X 0,Y 605.887,Z 843.44,A -85,B 0,C 180,E1 896.01,E2 896.01} C_VEL
LIN {X 0,Y 601.886,Z 843.44,A -85,B 0,C 180,E1 897.637,E2 897.637} C_VEL
LIN {X 0,Y 602.159,Z 843.44,A -85,B 0,C 180,E1 901.441,E2 901.441} C_VEL
LIN {X 0,Y 602.18,Z 843.44,A -85,B 0,C 180,E1 905.772,E2 905.772} C_VEL
LIN {X 0,Y 601.856,Z 843.44,A -85,B 0,C 180,E1 911.61,E2 911.61} C_VEL
LIN {X 0,Y 601.846,Z 843.44,A -85,B 0,C 180,E1 916.064,E2 916.064} C_VEL
LIN {X 0,Y 601.767,Z 843.44,A -85,B 0,C 180,E1 921.415,E2 921.415} C_VEL
LIN {X 0,Y 601.995,Z 843.44,A -85,B 0,C 180,E1 925.312,E2 925.312} C_VEL
LIN {X 0,Y 601.728,Z 843.44,A -85,B 0,C 180,E1 931.181,E2 931.181} C_VEL
LIN {X 0,Y 601.783,Z 843.44,A -85,B 0,C 180,E1 937.142,E2 937.142} C_VEL
LIN {X 0,Y 601.766,Z 843.44,A -85,B 0,C 180,E1 943.141,E2 943.141} C_VEL
LIN {X 0,Y 601.587,Z 843.44,A -85,B 0,C 180,E1 949.127,E2 949.127} C_VEL
LIN {X 0,Y 601.504,Z 843.44,A -85,B 0,C 180,E1 953.652,E2 953.652} C_VEL
LIN {X 0,Y 601.988,Z 843.44,A -85,B 0,C 180,E1 955.935,E2 955.935} C_VEL
LIN {X 0,Y 604.144,Z 852.801,A -85,B 0,C 180,E1 956.216,E2 956.216} C_VEL
LIN {X 0,Y 604.215,Z 910.713,A -85,B 0,C 180,E1 957.184,E2 957.184} C_VEL
LIN {X 0,Y 603.98,Z 951.161,A -85,B 0,C 180,E1 958.458,E2 958.458} C_VEL
LIN {X 0,Y 603.592,Z 990.662,A -85,B 0,C 180,E1 960.292,E2 960.292} C_VEL
LIN {X 0,Y 603.272,Z 1027.444,A -85,B 0,C 180,E1 962.605,E2 962.605} C_VEL
LIN {X 0,Y 602.849,Z 1062.042,A -85,B 0,C 180,E1 965.419,E2 965.419} C_VEL
LIN {X 0,Y 602.517,Z 1092.055,A -85,B 0,C 180,E1 968.523,E2 968.523} C_VEL
LIN {X 0,Y 602.263,Z 1118.926,A -85,B 0,C 180,E1 972.064,E2 972.064} C_VEL
LIN {X 0,Y 602.158,Z 1140.719,A -85,B 0,C 180,E1 975.809,E2 975.809} C_VEL
LIN {X 0,Y 602.062,Z 1156.737,A -85,B 0,C 180,E1 979.578,E2 979.578} C_VEL
LIN {X 0,Y 602.052,Z 1166.332,A -85,B 0,C 180,E1 982.777,E2 982.777} C_VEL
LIN {X 0,Y 602.172,Z 1171.905,A -85,B 0,C 180,E1 985.675,E2 985.675} C_VEL
LIN {X 0,Y 602.207,Z 1174.657,A -85,B 0,C 180,E1 988.56,E2 988.56} C_VEL
LIN {X 0,Y 602.081,Z 1173.626,A -85,B 0,C 180,E1 992.884,E2 992.884} C_VEL
LIN {X 0,Y 602.18,Z 1166.329,A -85,B 0,C 180,E1 997.223,E2 997.223} C_VEL
LIN {X 0,Y 602.106,Z 1153.525,A -85,B 0,C 180,E1 1001.295,E2 1001.295} C_VEL
LIN {X 0,Y 602.2,Z 1134.817,A -85,B 0,C 180,E1 1005.309,E2 1005.309} C_VEL
LIN {X 0,Y 602.338,Z 1111.002,A -85,B 0,C 180,E1 1009.075,E2 1009.075} C_VEL
LIN {X 0,Y 602.632,Z 1083,A -85,B 0,C 180,E1 1012.49,E2 1012.49} C_VEL
LIN {X 0,Y 602.982,Z 1050.171,A -85,B 0,C 180,E1 1015.629,E2 1015.629} C_VEL
LIN {X 0,Y 603.416,Z 1013.114,A -85,B 0,C 180,E1 1018.374,E2 1018.374} C_VEL
LIN {X 0,Y 603.796,Z 974.136,A -85,B 0,C 180,E1 1020.55,E2 1020.55} C_VEL
LIN {X 0,Y 604.149,Z 935.849,A -85,B 0,C 180,E1 1022.087,E2 1022.087} C_VEL
LIN {X 0,Y 604.344,Z 899.392,A -85,B 0,C 180,E1 1023.055,E2 1023.055} C_VEL
LIN {X 0,Y 603.531,Z 847.905,A -85,B 0,C 180,E1 1023.892,E2 1023.892} C_VEL
LIN {X 0,Y 602.106,Z 843.44,A -85,B 0,C 180,E1 1024.127,E2 1024.127} C_VEL
LIN {X 0,Y 601.742,Z 843.44,A -85,B 0,C 180,E1 1028.982,E2 1028.982} C_VEL
LIN {X 0,Y 601.599,Z 843.44,A -85,B 0,C 180,E1 1033.13,E2 1033.13} C_VEL
LIN {X 0,Y 601.736,Z 843.44,A -85,B 0,C 180,E1 1039.144,E2 1039.144} C_VEL
LIN {X 0,Y 601.874,Z 843.44,A -85,B 0,C 180,E1 1044.651,E2 1044.651} C_VEL
LIN {X 0,Y 601.75,Z 843.44,A -85,B 0,C 180,E1 1049.789,E2 1049.789} C_VEL
LIN {X 0,Y 601.734,Z 843.44,A -85,B 0,C 180,E1 1053.071,E2 1053.071} C_VEL
LIN {X 0,Y 601.564,Z 843.44,A -85,B 0,C 180,E1 1058.638,E2 1058.638} C_VEL
LIN {X 0,Y 601.066,Z 843.44,A -85,B 0,C 180,E1 1062.406,E2 1062.406} C_VEL
LIN {X 0,Y 602.828,Z 860.882,A -85,B 0,C 180,E1 1062.686,E2 1062.686} C_VEL
LIN {X 0,Y 602.763,Z 894.092,A -85,B 0,C 180,E1 1063.3,E2 1063.3} C_VEL
LIN {X 0,Y 602.72,Z 924.094,A -85,B 0,C 180,E1 1064.427,E2 1064.427} C_VEL
LIN {X 0,Y 602.541,Z 952.182,A -85,B 0,C 180,E1 1066.097,E2 1066.097} C_VEL
LIN {X 0,Y 602.436,Z 976.612,A -85,B 0,C 180,E1 1068.218,E2 1068.218} C_VEL
LIN {X 0,Y 602.285,Z 997.096,A -85,B 0,C 180,E1 1070.778,E2 1070.778} C_VEL
LIN {X 0,Y 602.251,Z 1011.729,A -85,B 0,C 180,E1 1073.507,E2 1073.507} C_VEL
LIN {X 0,Y 602.198,Z 1021.032,A -85,B 0,C 180,E1 1076.396,E2 1076.396} C_VEL
LIN {X 0,Y 602.183,Z 1024.384,A -85,B 0,C 180,E1 1078.559,E2 1078.559} C_VEL
LIN {X 0,Y 602.178,Z 1024.317,A -85,B 0,C 180,E1 1081.44,E2 1081.44} C_VEL
LIN {X 0,Y 602.224,Z 1019.008,A -85,B 0,C 180,E1 1084.325,E2 1084.325} C_VEL
LIN {X 0,Y 602.249,Z 1008.005,A -85,B 0,C 180,E1 1087.22,E2 1087.22} C_VEL
LIN {X 0,Y 602.341,Z 991.378,A -85,B 0,C 180,E1 1089.95,E2 1089.95} C_VEL
LIN {X 0,Y 602.431,Z 970.146,A -85,B 0,C 180,E1 1092.333,E2 1092.333} C_VEL
LIN {X 0,Y 602.629,Z 944.16,A -85,B 0,C 180,E1 1094.363,E2 1094.363} C_VEL
LIN {X 0,Y 602.778,Z 914.848,A -85,B 0,C 180,E1 1095.897,E2 1095.897} C_VEL
LIN {X 0,Y 602.846,Z 883.355,A -85,B 0,C 180,E1 1096.875,E2 1096.875} C_VEL
LIN {X 0,Y 602.112,Z 843.44,A -85,B 0,C 180,E1 1097.496,E2 1097.496} C_VEL
LIN {X 0,Y 601.74,Z 843.44,A -85,B 0,C 180,E1 1103.737,E2 1103.737} C_VEL
LIN {X 0,Y 601.781,Z 843.44,A -85,B 0,C 180,E1 1108.554,E2 1108.554} C_VEL
LIN {X 0,Y 601.913,Z 843.44,A -85,B 0,C 180,E1 1113.887,E2 1113.887} C_VEL
LIN {X 0,Y 601.719,Z 843.44,A -85,B 0,C 180,E1 1118.976,E2 1118.976} C_VEL
LIN {X 0,Y 601.579,Z 843.44,A -85,B 0,C 180,E1 1123.12,E2 1123.12} C_VEL
LIN {X 0,Y 601.74,Z 843.44,A -85,B 0,C 180,E1 1129.138,E2 1129.138} C_VEL
LIN {X 0,Y 601.923,Z 843.44,A -85,B 0,C 180,E1 1134.65,E2 1134.65} C_VEL
LIN {X 0,Y 602.086,Z 843.596,A -85,B 0,C 180,E1 1140.143,E2 1140.143} C_VEL
LIN {X 0,Y 603.282,Z 854.686,A -85,B 0,C 180,E1 1140.357,E2 1140.357} C_VEL
LIN {X 0,Y 603.796,Z 911.664,A -85,B 0,C 180,E1 1141.284,E2 1141.284} C_VEL
LIN {X 0,Y 603.584,Z 951.809,A -85,B 0,C 180,E1 1142.541,E2 1142.541} C_VEL
LIN {X 0,Y 603.294,Z 989.566,A -85,B 0,C 180,E1 1144.346,E2 1144.346} C_VEL
LIN {X 0,Y 602.964,Z 1024.255,A -85,B 0,C 180,E1 1146.63,E2 1146.63} C_VEL
LIN {X 0,Y 602.635,Z 1056.168,A -85,B 0,C 180,E1 1149.405,E2 1149.405} C_VEL
LIN {X 0,Y 602.405,Z 1083.068,A -85,B 0,C 180,E1 1152.445,E2 1152.445} C_VEL
LIN {X 0,Y 602.273,Z 1105.82,A -85,B 0,C 180,E1 1155.811,E2 1155.811} C_VEL
LIN {X 0,Y 602.169,Z 1123.128,A -85,B 0,C 180,E1 1159.276,E2 1159.276} C_VEL
LIN {X 0,Y 602.11,Z 1135.23,A -85,B 0,C 180,E1 1162.776,E2 1162.776} C_VEL
LIN {X 0,Y 602.055,Z 1141.505,A -85,B 0,C 180,E1 1165.672,E2 1165.672} C_VEL
LIN {X 0,Y 602.042,Z 1144.613,A -85,B 0,C 180,E1 1168.558,E2 1168.558} C_VEL
LIN {X 0,Y 602.19,Z 1144.551,A -85,B 0,C 180,E1 1171.44,E2 1171.44} C_VEL
LIN {X 0,Y 602.216,Z 1140.139,A -85,B 0,C 180,E1 1175.048,E2 1175.048} C_VEL
LIN {X 0,Y 602.201,Z 1129.296,A -85,B 0,C 180,E1 1179.041,E2 1179.041} C_VEL
LIN {X 0,Y 602.245,Z 1113.482,A -85,B 0,C 180,E1 1182.708,E2 1182.708} C_VEL
LIN {X 0,Y 602.356,Z 1092.405,A -85,B 0,C 180,E1 1186.2,E2 1186.2} C_VEL
LIN {X 0,Y 602.58,Z 1066.205,A -85,B 0,C 180,E1 1189.46,E2 1189.46} C_VEL
LIN {X 0,Y 602.821,Z 1036.417,A -85,B 0,C 180,E1 1192.309,E2 1192.309} C_VEL
LIN {X 0,Y 603.15,Z 1002.853,A -85,B 0,C 180,E1 1194.766,E2 1194.766} C_VEL
LIN {X 0,Y 603.492,Z 966.366,A -85,B 0,C 180,E1 1196.746,E2 1196.746} C_VEL
LIN {X 0,Y 603.755,Z 927.514,A -85,B 0,C 180,E1 1198.201,E2 1198.201} C_VEL
LIN {X 0,Y 603.841,Z 889.371,A -85,B 0,C 180,E1 1199.048,E2 1199.048} C_VEL
LIN {X 0,Y 602.799,Z 847.366,A -85,B 0,C 180,E1 1199.677,E2 1199.677} C_VEL
LIN {X 0,Y 602.168,Z 843.44,A -85,B 0,C 180,E1 1199.831,E2 1199.831} C_VEL
LIN {X 0,Y 601.888,Z 843.44,A -85,B 0,C 180,E1 1207.138,E2 1207.138} C_VEL
LIN {X 0,Y 601.631,Z 843.44,A -85,B 0,C 180,E1 1213.135,E2 1213.135} C_VEL
LIN {X 0,Y 601.791,Z 843.44,A -85,B 0,C 180,E1 1217.216,E2 1217.216} C_VEL
LIN {X 0,Y 601.78,Z 843.44,A -85,B 0,C 180,E1 1223.624,E2 1223.624} C_VEL
LIN {X 0,Y 601.815,Z 843.44,A -85,B 0,C 180,E1 1229.794,E2 1229.794} C_VEL
LIN {X 0,Y 602.055,Z 843.44,A -85,B 0,C 180,E1 1234.873,E2 1234.873} C_VEL
LIN {X 0,Y 601.989,Z 843.44,A -85,B 0,C 180,E1 1240.918,E2 1240.918} C_VEL
LIN {X 0,Y 602.131,Z 843.44,A -85,B 0,C 180,E1 1246.922,E2 1246.922} C_VEL
LIN {X 0,Y 601.918,Z 843.44,A -85,B 0,C 180,E1 1252.776,E2 1252.776} C_VEL
LIN {X 0,Y 601.886,Z 843.44,A -85,B 0,C 180,E1 1257.637,E2 1257.637} C_VEL
LIN {X 0,Y 597.831,Z 843.44,A -85,B 0,C 180,E1 1259.261,E2 1259.261} C_VEL
LIN {X 0,Y 594.111,Z 843.44,A -85,B 0,C 180,E1 1260.907,E2 1260.907} C_VEL
LIN {X 0,Y 594.117,Z 843.44,A -85,B 0,C 180,E1 1266.321,E2 1266.321} C_VEL
LIN {X 0,Y 593.92,Z 843.44,A -85,B 0,C 180,E1 1271.767,E2 1271.767} C_VEL
LIN {X 0,Y 593.901,Z 843.44,A -85,B 0,C 180,E1 1276.285,E2 1276.285} C_VEL
LIN {X 0,Y 593.988,Z 843.44,A -85,B 0,C 180,E1 1280.906,E2 1280.906} C_VEL
LIN {X 0,Y 593.982,Z 843.44,A -85,B 0,C 180,E1 1285.678,E2 1285.678} C_VEL
LIN {X 0,Y 593.876,Z 843.44,A -85,B 0,C 180,E1 1290.655,E2 1290.655} C_VEL
LIN {X 0,Y 593.862,Z 843.44,A -85,B 0,C 180,E1 1295.899,E2 1295.899} C_VEL
LIN {X 0,Y 593.789,Z 843.44,A -85,B 0,C 180,E1 1301.523,E2 1301.523} C_VEL
LIN {X 0,Y 593.726,Z 843.44,A -85,B 0,C 180,E1 1306.485,E2 1306.485} C_VEL
LIN {X 0,Y 593.709,Z 843.44,A -85,B 0,C 180,E1 1312.261,E2 1312.261} C_VEL
LIN {X 0,Y 593.896,Z 843.712,A -85,B 0,C 180,E1 1315.421,E2 1315.421} C_VEL
LIN {X 0,Y 597.616,Z 854.541,A -85,B 0,C 180,E1 1315.821,E2 1315.821} C_VEL
LIN {X 0,Y 597.557,Z 910.642,A -85,B 0,C 180,E1 1316.77,E2 1316.77} C_VEL
LIN {X 0,Y 597.189,Z 951.165,A -85,B 0,C 180,E1 1318.057,E2 1318.057} C_VEL
LIN {X 0,Y 596.573,Z 989.612,A -85,B 0,C 180,E1 1319.848,E2 1319.848} C_VEL
LIN {X 0,Y 596.011,Z 1027.074,A -85,B 0,C 180,E1 1322.215,E2 1322.215} C_VEL
LIN {X 0,Y 595.377,Z 1061.874,A -85,B 0,C 180,E1 1325.074,E2 1325.074} C_VEL
LIN {X 0,Y 594.879,Z 1092.056,A -85,B 0,C 180,E1 1328.233,E2 1328.233} C_VEL
LIN {X 0,Y 594.515,Z 1118.928,A -85,B 0,C 180,E1 1331.822,E2 1331.822} C_VEL
LIN {X 0,Y 594.316,Z 1139.96,A -85,B 0,C 180,E1 1335.469,E2 1335.469} C_VEL
LIN {X 0,Y 594.192,Z 1155.953,A -85,B 0,C 180,E1 1339.222,E2 1339.222} C_VEL
LIN {X 0,Y 594.162,Z 1166.332,A -85,B 0,C 180,E1 1342.68,E2 1342.68} C_VEL
LIN {X 0,Y 594.276,Z 1171.905,A -85,B 0,C 180,E1 1345.617,E2 1345.617} C_VEL
LIN {X 0,Y 594.3,Z 1174.657,A -85,B 0,C 180,E1 1348.541,E2 1348.541} C_VEL
LIN {X 0,Y 594.175,Z 1173.626,A -85,B 0,C 180,E1 1352.922,E2 1352.922} C_VEL
LIN {X 0,Y 594.293,Z 1166.329,A -85,B 0,C 180,E1 1357.319,E2 1357.319} C_VEL
LIN {X 0,Y 594.224,Z 1154.015,A -85,B 0,C 180,E1 1361.312,E2 1361.312} C_VEL
LIN {X 0,Y 594.396,Z 1136.79,A -85,B 0,C 180,E1 1365.136,E2 1365.136} C_VEL
LIN {X 0,Y 594.614,Z 1115.029,A -85,B 0,C 180,E1 1368.753,E2 1368.753} C_VEL
LIN {X 0,Y 595.001,Z 1087.602,A -85,B 0,C 180,E1 1372.279,E2 1372.279} C_VEL
LIN {X 0,Y 595.49,Z 1055.718,A -85,B 0,C 180,E1 1375.485,E2 1375.485} C_VEL
LIN {X 0,Y 596.142,Z 1020.242,A -85,B 0,C 180,E1 1378.266,E2 1378.266} C_VEL
LIN {X 0,Y 596.731,Z 981.765,A -85,B 0,C 180,E1 1380.57,E2 1380.57} C_VEL
LIN {X 0,Y 597.344,Z 941.168,A -85,B 0,C 180,E1 1382.318,E2 1382.318} C_VEL
LIN {X 0,Y 597.679,Z 901.59,A -85,B 0,C 180,E1 1383.423,E2 1383.423} C_VEL
LIN {X 0,Y 596.92,Z 850.575,A -85,B 0,C 180,E1 1384.281,E2 1384.281} C_VEL
LIN {X 0,Y 594.141,Z 843.44,A -85,B 0,C 180,E1 1384.596,E2 1384.596} C_VEL
LIN {X 0,Y 593.77,Z 843.44,A -85,B 0,C 180,E1 1390.1,E2 1390.1} C_VEL
LIN {X 0,Y 593.55,Z 843.44,A -85,B 0,C 180,E1 1395.585,E2 1395.585} C_VEL
LIN {X 0,Y 593.774,Z 843.44,A -85,B 0,C 180,E1 1400.399,E2 1400.399} C_VEL
LIN {X 0,Y 594.005,Z 843.44,A -85,B 0,C 180,E1 1405.894,E2 1405.894} C_VEL
LIN {X 0,Y 593.994,Z 843.44,A -85,B 0,C 180,E1 1411.035,E2 1411.035} C_VEL
LIN {X 0,Y 593.787,Z 843.44,A -85,B 0,C 180,E1 1416.635,E2 1416.635} C_VEL
LIN {X 0,Y 593.694,Z 843.44,A -85,B 0,C 180,E1 1420.673,E2 1420.673} C_VEL
LIN {X 0,Y 593.227,Z 843.44,A -85,B 0,C 180,E1 1422.166,E2 1422.166} C_VEL
LIN {X 0,Y 595.292,Z 860.531,A -85,B 0,C 180,E1 1422.456,E2 1422.456} C_VEL
LIN {X 0,Y 595.193,Z 894.063,A -85,B 0,C 180,E1 1423.081,E2 1423.081} C_VEL
LIN {X 0,Y 595.044,Z 924.087,A -85,B 0,C 180,E1 1424.221,E2 1424.221} C_VEL
LIN {X 0,Y 594.799,Z 952.375,A -85,B 0,C 180,E1 1425.928,E2 1425.928} C_VEL
LIN {X 0,Y 594.617,Z 976.61,A -85,B 0,C 180,E1 1428.06,E2 1428.06} C_VEL
LIN {X 0,Y 594.437,Z 997.095,A -85,B 0,C 180,E1 1430.655,E2 1430.655} C_VEL
LIN {X 0,Y 594.363,Z 1011.981,A -85,B 0,C 180,E1 1433.48,E2 1433.48} C_VEL
LIN {X 0,Y 594.307,Z 1021.033,A -85,B 0,C 180,E1 1436.348,E2 1436.348} C_VEL
LIN {X 0,Y 594.281,Z 1024.386,A -85,B 0,C 180,E1 1438.54,E2 1438.54} C_VEL
LIN {X 0,Y 594.276,Z 1024.317,A -85,B 0,C 180,E1 1441.459,E2 1441.459} C_VEL
LIN {X 0,Y 594.322,Z 1019.011,A -85,B 0,C 180,E1 1444.382,E2 1444.382} C_VEL
LIN {X 0,Y 594.373,Z 1008.009,A -85,B 0,C 180,E1 1447.316,E2 1447.316} C_VEL
LIN {X 0,Y 594.475,Z 991.386,A -85,B 0,C 180,E1 1450.083,E2 1450.083} C_VEL
LIN {X 0,Y 594.644,Z 970.156,A -85,B 0,C 180,E1 1452.497,E2 1452.497} C_VEL
LIN {X 0,Y 594.912,Z 944.205,A -85,B 0,C 180,E1 1454.551,E2 1454.551} C_VEL
LIN {X 0,Y 595.165,Z 914.862,A -85,B 0,C 180,E1 1456.106,E2 1456.106} C_VEL
LIN {X 0,Y 595.279,Z 883.364,A -85,B 0,C 180,E1 1457.096,E2 1457.096} C_VEL
LIN {X 0,Y 594.621,Z 846.101,A -85,B 0,C 180,E1 1457.654,E2 1457.654} C_VEL
LIN {X 0,Y 594.118,Z 843.44,A -85,B 0,C 180,E1 1457.751,E2 1457.751} C_VEL
LIN {X 0,Y 593.804,Z 843.44,A -85,B 0,C 180,E1 1464.074,E2 1464.074} C_VEL
LIN {X 0,Y 593.784,Z 843.44,A -85,B 0,C 180,E1 1468.975,E2 1468.975} C_VEL
LIN {X 0,Y 593.99,Z 843.44,A -85,B 0,C 180,E1 1474.105,E2 1474.105} C_VEL
LIN {X 0,Y 593.734,Z 843.44,A -85,B 0,C 180,E1 1480.087,E2 1480.087} C_VEL
LIN {X 0,Y 593.541,Z 843.44,A -85,B 0,C 180,E1 1485.576,E2 1485.576} C_VEL
LIN {X 0,Y 593.77,Z 843.44,A -85,B 0,C 180,E1 1490.393,E2 1490.393} C_VEL
LIN {X 0,Y 594.079,Z 843.44,A -85,B 0,C 180,E1 1495.894,E2 1495.894} C_VEL
LIN {X 0,Y 594.091,Z 843.44,A -85,B 0,C 180,E1 1499.693,E2 1499.693} C_VEL
LIN {X 0,Y 596.383,Z 851.653,A -85,B 0,C 180,E1 1499.939,E2 1499.939} C_VEL
LIN {X 0,Y 596.832,Z 912.116,A -85,B 0,C 180,E1 1500.929,E2 1500.929} C_VEL
LIN {X 0,Y 596.474,Z 952.52,A -85,B 0,C 180,E1 1502.217,E2 1502.217} C_VEL
LIN {X 0,Y 596.014,Z 990.707,A -85,B 0,C 180,E1 1504.078,E2 1504.078} C_VEL
LIN {X 0,Y 595.491,Z 1025.299,A -85,B 0,C 180,E1 1506.402,E2 1506.402} C_VEL
LIN {X 0,Y 595.008,Z 1056.162,A -85,B 0,C 180,E1 1509.128,E2 1509.128} C_VEL
LIN {X 0,Y 594.675,Z 1083.064,A -85,B 0,C 180,E1 1512.209,E2 1512.209} C_VEL
LIN {X 0,Y 594.413,Z 1104.703,A -85,B 0,C 180,E1 1515.427,E2 1515.427} C_VEL
LIN {X 0,Y 594.29,Z 1122.341,A -85,B 0,C 180,E1 1518.944,E2 1518.944} C_VEL
LIN {X 0,Y 594.226,Z 1135.228,A -85,B 0,C 180,E1 1522.68,E2 1522.68} C_VEL
LIN {X 0,Y 594.151,Z 1141.505,A -85,B 0,C 180,E1 1525.615,E2 1525.615} C_VEL
LIN {X 0,Y 594.141,Z 1144.613,A -85,B 0,C 180,E1 1528.539,E2 1528.539} C_VEL
LIN {X 0,Y 594.285,Z 1144.552,A -85,B 0,C 180,E1 1531.459,E2 1531.459} C_VEL
LIN {X 0,Y 594.329,Z 1140.14,A -85,B 0,C 180,E1 1535.115,E2 1535.115} C_VEL
LIN {X 0,Y 594.305,Z 1129.298,A -85,B 0,C 180,E1 1539.162,E2 1539.162} C_VEL
LIN {X 0,Y 594.395,Z 1113.486,A -85,B 0,C 180,E1 1542.878,E2 1542.878} C_VEL
LIN {X 0,Y 594.583,Z 1093.472,A -85,B 0,C 180,E1 1546.267,E2 1546.267} C_VEL
LIN {X 0,Y 594.881,Z 1067.947,A -85,B 0,C 180,E1 1549.531,E2 1549.531} C_VEL
LIN {X 0,Y 595.299,Z 1038.5,A -85,B 0,C 180,E1 1552.427,E2 1552.427} C_VEL
LIN {X 0,Y 595.791,Z 1005.114,A -85,B 0,C 180,E1 1554.944,E2 1554.944} C_VEL
LIN {X 0,Y 596.284,Z 969.557,A -85,B 0,C 180,E1 1556.942,E2 1556.942} C_VEL
LIN {X 0,Y 596.673,Z 932.187,A -85,B 0,C 180,E1 1558.419,E2 1558.419} C_VEL
LIN {X 0,Y 596.915,Z 893.141,A -85,B 0,C 180,E1 1559.358,E2 1559.358} C_VEL
LIN {X 0,Y 596.012,Z 848.917,A -85,B 0,C 180,E1 1560.029,E2 1560.029} C_VEL
LIN {X 0,Y 594.1,Z 843.44,A -85,B 0,C 180,E1 1560.286,E2 1560.286} C_VEL
LIN {X 0,Y 593.892,Z 843.44,A -85,B 0,C 180,E1 1565.9,E2 1565.9} C_VEL
LIN {X 0,Y 593.648,Z 843.44,A -85,B 0,C 180,E1 1571.539,E2 1571.539} C_VEL
LIN {X 0,Y 593.832,Z 843.44,A -85,B 0,C 180,E1 1576.501,E2 1576.501} C_VEL
LIN {X 0,Y 593.771,Z 843.44,A -85,B 0,C 180,E1 1582.272,E2 1582.272} C_VEL
LIN {X 0,Y 593.64,Z 843.44,A -85,B 0,C 180,E1 1587.619,E2 1587.619} C_VEL
LIN {X 0,Y 593.74,Z 843.44,A -85,B 0,C 180,E1 1592.68,E2 1592.68} C_VEL
LIN {X 0,Y 593.764,Z 843.44,A -85,B 0,C 180,E1 1597.515,E2 1597.515} C_VEL
LIN {X 0,Y 593.992,Z 843.44,A -85,B 0,C 180,E1 1602.191,E2 1602.191} C_VEL
LIN {X 0,Y 594.192,Z 843.44,A -85,B 0,C 180,E1 1606.744,E2 1606.744} C_VEL
LIN {X 0,Y 594.026,Z 843.44,A -85,B 0,C 180,E1 1612.68,E2 1612.68} C_VEL
LIN {X 0,Y 593.98,Z 843.44,A -85,B 0,C 180,E1 1617.622,E2 1617.622} C_VEL
LIN {X 0,Y 594.111,Z 843.44,A -85,B 0,C 180,E1 1620.907,E2 1620.907} C_VEL
LIN {X 0,Y 591.604,Z 843.44,A -85,B 0,C 180,E1 1622.151,E2 1622.151} C_VEL
LIN {X 0,Y 586.093,Z 843.44,A -85,B 0,C 180,E1 1624.011,E2 1624.011} C_VEL
LIN {X 0,Y 586.016,Z 843.44,A -85,B 0,C 180,E1 1624.226,E2 1624.226} C_VEL
LIN {X 0,Y 585.95,Z 843.44,A -85,B 0,C 180,E1 1628.919,E2 1628.919} C_VEL
LIN {X 0,Y 585.957,Z 843.44,A -85,B 0,C 180,E1 1633.447,E2 1633.447} C_VEL
LIN {X 0,Y 585.882,Z 843.44,A -85,B 0,C 180,E1 1638.065,E2 1638.065} C_VEL
LIN {X 0,Y 585.892,Z 843.44,A -85,B 0,C 180,E1 1642.806,E2 1642.806} C_VEL
LIN {X 0,Y 585.814,Z 843.44,A -85,B 0,C 180,E1 1647.723,E2 1647.723} C_VEL
LIN {X 0,Y 585.74,Z 843.44,A -85,B 0,C 180,E1 1652.874,E2 1652.874} C_VEL
LIN {X 0,Y 585.859,Z 843.44,A -85,B 0,C 180,E1 1658.331,E2 1658.331} C_VEL
LIN {X 0,Y 585.915,Z 843.44,A -85,B 0,C 180,E1 1664.24,E2 1664.24} C_VEL
LIN {X 0,Y 585.802,Z 843.44,A -85,B 0,C 180,E1 1669.747,E2 1669.747} C_VEL
LIN {X 0,Y 585.859,Z 843.715,A -85,B 0,C 180,E1 1674.878,E2 1674.878} C_VEL
LIN {X 0,Y 591,Z 854.75,A -85,B 0,C 180,E1 1675.387,E2 1675.387} C_VEL
LIN {X 0,Y 590.922,Z 910.887,A -85,B 0,C 180,E1 1676.353,E2 1676.353} C_VEL
LIN {X 0,Y 590.382,Z 951.803,A -85,B 0,C 180,E1 1677.669,E2 1677.669} C_VEL
LIN {X 0,Y 589.622,Z 989.616,A -85,B 0,C 180,E1 1679.455,E2 1679.455} C_VEL
LIN {X 0,Y 588.798,Z 1025.907,A -85,B 0,C 180,E1 1681.756,E2 1681.756} C_VEL
LIN {X 0,Y 587.955,Z 1061.832,A -85,B 0,C 180,E1 1684.733,E2 1684.733} C_VEL
LIN {X 0,Y 587.253,Z 1092.825,A -85,B 0,C 180,E1 1688.03,E2 1688.03} C_VEL
LIN {X 0,Y 586.753,Z 1118.929,A -85,B 0,C 180,E1 1691.573,E2 1691.573} C_VEL
LIN {X 0,Y 586.48,Z 1140.624,A -85,B 0,C 180,E1 1695.402,E2 1695.402} C_VEL
LIN {X 0,Y 586.336,Z 1156.504,A -85,B 0,C 180,E1 1699.229,E2 1699.229} C_VEL
LIN {X 0,Y 586.276,Z 1166.332,A -85,B 0,C 180,E1 1702.581,E2 1702.581} C_VEL
LIN {X 0,Y 586.38,Z 1171.905,A -85,B 0,C 180,E1 1705.558,E2 1705.558} C_VEL
LIN {X 0,Y 586.395,Z 1174.657,A -85,B 0,C 180,E1 1708.521,E2 1708.521} C_VEL
LIN {X 0,Y 586.277,Z 1173.626,A -85,B 0,C 180,E1 1712.961,E2 1712.961} C_VEL
LIN {X 0,Y 586.38,Z 1166.329,A -85,B 0,C 180,E1 1717.419,E2 1717.419} C_VEL
LIN {X 0,Y 586.355,Z 1154.015,A -85,B 0,C 180,E1 1721.466,E2 1721.466} C_VEL
LIN {X 0,Y 586.535,Z 1136.792,A -85,B 0,C 180,E1 1725.344,E2 1725.344} C_VEL
LIN {X 0,Y 586.864,Z 1115.031,A -85,B 0,C 180,E1 1729.011,E2 1729.011} C_VEL
LIN {X 0,Y 587.417,Z 1087.268,A -85,B 0,C 180,E1 1732.62,E2 1732.62} C_VEL
LIN {X 0,Y 588.108,Z 1055.705,A -85,B 0,C 180,E1 1735.83,E2 1735.83} C_VEL
LIN {X 0,Y 588.913,Z 1020.651,A -85,B 0,C 180,E1 1738.617,E2 1738.617} C_VEL
LIN {X 0,Y 589.798,Z 981.649,A -85,B 0,C 180,E1 1740.975,E2 1740.975} C_VEL
LIN {X 0,Y 590.607,Z 941.165,A -85,B 0,C 180,E1 1742.733,E2 1742.733} C_VEL
LIN {X 0,Y 591.07,Z 901.961,A -85,B 0,C 180,E1 1743.839,E2 1743.839} C_VEL
LIN {X 0,Y 590.437,Z 853.257,A -85,B 0,C 180,E1 1744.672,E2 1744.672} C_VEL
LIN {X 0,Y 586.171,Z 843.44,A -85,B 0,C 180,E1 1745.126,E2 1745.126} C_VEL
LIN {X 0,Y 585.865,Z 843.44,A -85,B 0,C 180,E1 1751.461,E2 1751.461} C_VEL
LIN {X 0,Y 585.845,Z 843.44,A -85,B 0,C 180,E1 1757.786,E2 1757.786} C_VEL
LIN {X 0,Y 585.937,Z 843.44,A -85,B 0,C 180,E1 1763.538,E2 1763.538} C_VEL
LIN {X 0,Y 585.886,Z 843.44,A -85,B 0,C 180,E1 1768.523,E2 1768.523} C_VEL
LIN {X 0,Y 585.857,Z 843.44,A -85,B 0,C 180,E1 1773.94,E2 1773.94} C_VEL
LIN {X 0,Y 585.719,Z 843.44,A -85,B 0,C 180,E1 1778.784,E2 1778.784} C_VEL
LIN {X 0,Y 585.375,Z 843.44,A -85,B 0,C 180,E1 1781.919,E2 1781.919} C_VEL
LIN {X 0,Y 587.781,Z 860.007,A -85,B 0,C 180,E1 1782.218,E2 1782.218} C_VEL
LIN {X 0,Y 587.631,Z 894.08,A -85,B 0,C 180,E1 1782.858,E2 1782.858} C_VEL
LIN {X 0,Y 587.43,Z 924.08,A -85,B 0,C 180,E1 1784.011,E2 1784.011} C_VEL
LIN {X 0,Y 587.074,Z 952.563,A -85,B 0,C 180,E1 1785.754,E2 1785.754} C_VEL
LIN {X 0,Y 586.818,Z 976.608,A -85,B 0,C 180,E1 1787.899,E2 1787.899} C_VEL
LIN {X 0,Y 586.594,Z 997.093,A -85,B 0,C 180,E1 1790.529,E2 1790.529} C_VEL
LIN {X 0,Y 586.466,Z 1011.98,A -85,B 0,C 180,E1 1793.392,E2 1793.392} C_VEL
LIN {X 0,Y 586.424,Z 1021.033,A -85,B 0,C 180,E1 1796.299,E2 1796.299} C_VEL
LIN {X 0,Y 586.386,Z 1024.388,A -85,B 0,C 180,E1 1798.52,E2 1798.52} C_VEL
LIN {X 0,Y 586.381,Z 1024.316,A -85,B 0,C 180,E1 1801.479,E2 1801.479} C_VEL
LIN {X 0,Y 586.423,Z 1019.014,A -85,B 0,C 180,E1 1804.441,E2 1804.441} C_VEL
LIN {X 0,Y 586.481,Z 1008.014,A -85,B 0,C 180,E1 1807.415,E2 1807.415} C_VEL
LIN {X 0,Y 586.633,Z 991.393,A -85,B 0,C 180,E1 1810.219,E2 1810.219} C_VEL
LIN {X 0,Y 586.857,Z 970.166,A -85,B 0,C 180,E1 1812.666,E2 1812.666} C_VEL
LIN {X 0,Y 587.199,Z 944.214,A -85,B 0,C 180,E1 1814.747,E2 1814.747} C_VEL
LIN {X 0,Y 587.545,Z 914.875,A -85,B 0,C 180,E1 1816.321,E2 1816.321} C_VEL
LIN {X 0,Y 587.718,Z 883.822,A -85,B 0,C 180,E1 1817.313,E2 1817.313} C_VEL
LIN {X 0,Y 586.956,Z 846.897,A -85,B 0,C 180,E1 1817.883,E2 1817.883} C_VEL
LIN {X 0,Y 586.117,Z 843.44,A -85,B 0,C 180,E1 1818.002,E2 1818.002} C_VEL
LIN {X 0,Y 585.958,Z 843.44,A -85,B 0,C 180,E1 1822.802,E2 1822.802} C_VEL
LIN {X 0,Y 585.852,Z 843.44,A -85,B 0,C 180,E1 1828.509,E2 1828.509} C_VEL
LIN {X 0,Y 586.034,Z 843.44,A -85,B 0,C 180,E1 1834.634,E2 1834.634} C_VEL
LIN {X 0,Y 585.846,Z 843.44,A -85,B 0,C 180,E1 1840.243,E2 1840.243} C_VEL
LIN {X 0,Y 585.723,Z 843.44,A -85,B 0,C 180,E1 1846.362,E2 1846.362} C_VEL
LIN {X 0,Y 585.893,Z 843.44,A -85,B 0,C 180,E1 1851.666,E2 1851.666} C_VEL
LIN {X 0,Y 586.121,Z 843.44,A -85,B 0,C 180,E1 1857.145,E2 1857.145} C_VEL
LIN {X 0,Y 586.141,Z 843.44,A -85,B 0,C 180,E1 1859.222,E2 1859.222} C_VEL
LIN {X 0,Y 589.561,Z 854.596,A -85,B 0,C 180,E1 1859.596,E2 1859.596} C_VEL
LIN {X 0,Y 589.93,Z 912.226,A -85,B 0,C 180,E1 1860.56,E2 1860.56} C_VEL
LIN {X 0,Y 589.431,Z 952,A -85,B 0,C 180,E1 1861.834,E2 1861.834} C_VEL
LIN {X 0,Y 588.771,Z 990.073,A -85,B 0,C 180,E1 1863.698,E2 1863.698} C_VEL
LIN {X 0,Y 588.042,Z 1025.293,A -85,B 0,C 180,E1 1866.084,E2 1866.084} C_VEL
LIN {X 0,Y 587.424,Z 1056.156,A -85,B 0,C 180,E1 1868.846,E2 1868.846} C_VEL
LIN {X 0,Y 586.936,Z 1083.06,A -85,B 0,C 180,E1 1871.966,E2 1871.966} C_VEL
LIN {X 0,Y 586.59,Z 1105.417,A -85,B 0,C 180,E1 1875.354,E2 1875.354} C_VEL
LIN {X 0,Y 586.418,Z 1122.449,A -85,B 0,C 180,E1 1878.82,E2 1878.82} C_VEL
LIN {X 0,Y 586.328,Z 1135.227,A -85,B 0,C 180,E1 1882.581,E2 1882.581} C_VEL
LIN {X 0,Y 586.248,Z 1141.504,A -85,B 0,C 180,E1 1885.555,E2 1885.555} C_VEL
LIN {X 0,Y 586.248,Z 1144.613,A -85,B 0,C 180,E1 1888.519,E2 1888.519} C_VEL
LIN {X 0,Y 586.381,Z 1144.552,A -85,B 0,C 180,E1 1891.479,E2 1891.479} C_VEL
LIN {X 0,Y 586.427,Z 1140.141,A -85,B 0,C 180,E1 1895.184,E2 1895.184} C_VEL
LIN {X 0,Y 586.454,Z 1130.572,A -85,B 0,C 180,E1 1898.911,E2 1898.911} C_VEL
LIN {X 0,Y 586.548,Z 1115.373,A -85,B 0,C 180,E1 1902.674,E2 1902.674} C_VEL
LIN {X 0,Y 586.801,Z 1093.474,A -85,B 0,C 180,E1 1906.489,E2 1906.489} C_VEL
LIN {X 0,Y 587.216,Z 1068.241,A -85,B 0,C 180,E1 1909.764,E2 1909.764} C_VEL
LIN {X 0,Y 587.783,Z 1038.509,A -85,B 0,C 180,E1 1912.73,E2 1912.73} C_VEL
LIN {X 0,Y 588.458,Z 1005.153,A -85,B 0,C 180,E1 1915.275,E2 1915.275} C_VEL
LIN {X 0,Y 589.132,Z 970.336,A -85,B 0,C 180,E1 1917.259,E2 1917.259} C_VEL
LIN {X 0,Y 589.662,Z 933.435,A -85,B 0,C 180,E1 1918.749,E2 1918.749} C_VEL
LIN {X 0,Y 590.017,Z 894.834,A -85,B 0,C 180,E1 1919.709,E2 1919.709} C_VEL
LIN {X 0,Y 589.309,Z 851.815,A -85,B 0,C 180,E1 1920.367,E2 1920.367} C_VEL
LIN {X 0,Y 586.088,Z 843.44,A -85,B 0,C 180,E1 1920.734,E2 1920.734} C_VEL
LIN {X 0,Y 585.963,Z 843.44,A -85,B 0,C 180,E1 1926.781,E2 1926.781} C_VEL
LIN {X 0,Y 585.749,Z 843.44,A -85,B 0,C 180,E1 1932.227,E2 1932.227} C_VEL
LIN {X 0,Y 585.914,Z 843.44,A -85,B 0,C 180,E1 1937.794,E2 1937.794} C_VEL
LIN {X 0,Y 585.845,Z 843.44,A -85,B 0,C 180,E1 1943.533,E2 1943.533} C_VEL
LIN {X 0,Y 585.856,Z 843.44,A -85,B 0,C 180,E1 1948.881,E2 1948.881} C_VEL
LIN {X 0,Y 586.035,Z 843.44,A -85,B 0,C 180,E1 1954.726,E2 1954.726} C_VEL
LIN {X 0,Y 586.148,Z 843.44,A -85,B 0,C 180,E1 1960.381,E2 1960.381} C_VEL
LIN {X 0,Y 586.269,Z 843.44,A -85,B 0,C 180,E1 1966.562,E2 1966.562} C_VEL
LIN {X 0,Y 586.123,Z 843.44,A -85,B 0,C 180,E1 1972.58,E2 1972.58} C_VEL
LIN {X 0,Y 586.227,Z 843.44,A -85,B 0,C 180,E1 1977.04,E2 1977.04} C_VEL
LIN {X 0,Y 586.345,Z 843.44,A -85,B 0,C 180,E1 1981.48,E2 1981.48} C_VEL
LIN {X 0,Y 586.016,Z 843.44,A -85,B 0,C 180,E1 1984.226,E2 1984.226} C_VEL
LIN {X 0,Y 583.59,Z 843.44,A -85,B 0,C 180,E1 1985.49,E2 1985.49} C_VEL
LIN {X 0,Y 578.081,Z 843.44,A -85,B 0,C 180,E1 1987.599,E2 1987.599} C_VEL
LIN {X 0,Y 578.09,Z 843.44,A -85,B 0,C 180,E1 1992.094,E2 1992.094} C_VEL
LIN {X 0,Y 578.043,Z 843.44,A -85,B 0,C 180,E1 1996.745,E2 1996.745} C_VEL
LIN {X 0,Y 578.078,Z 843.44,A -85,B 0,C 180,E1 2001.51,E2 2001.51} C_VEL
LIN {X 0,Y 577.957,Z 843.44,A -85,B 0,C 180,E1 2007.036,E2 2007.036} C_VEL
LIN {X 0,Y 577.916,Z 843.44,A -85,B 0,C 180,E1 2011.597,E2 2011.597} C_VEL
LIN {X 0,Y 577.976,Z 843.44,A -85,B 0,C 180,E1 2017.047,E2 2017.047} C_VEL
LIN {X 0,Y 577.97,Z 843.44,A -85,B 0,C 180,E1 2022.926,E2 2022.926} C_VEL
LIN {X 0,Y 577.844,Z 843.44,A -85,B 0,C 180,E1 2029.075,E2 2029.075} C_VEL
LIN {X 0,Y 577.868,Z 843.44,A -85,B 0,C 180,E1 2034.309,E2 2034.309} C_VEL
LIN {X 0,Y 584.134,Z 857.078,A -85,B 0,C 180,E1 2034.955,E2 2034.955} C_VEL
LIN {X 0,Y 584.27,Z 912.438,A -85,B 0,C 180,E1 2035.961,E2 2035.961} C_VEL
LIN {X 0,Y 583.564,Z 954.594,A -85,B 0,C 180,E1 2037.356,E2 2037.356} C_VEL
LIN {X 0,Y 582.521,Z 993.454,A -85,B 0,C 180,E1 2039.263,E2 2039.263} C_VEL
LIN {X 0,Y 581.472,Z 1030.447,A -85,B 0,C 180,E1 2041.717,E2 2041.717} C_VEL
LIN {X 0,Y 580.471,Z 1063.816,A -85,B 0,C 180,E1 2044.58,E2 2044.58} C_VEL
LIN {X 0,Y 579.605,Z 1093.769,A -85,B 0,C 180,E1 2047.843,E2 2047.843} C_VEL
LIN {X 0,Y 578.99,Z 1119.046,A -85,B 0,C 180,E1 2051.335,E2 2051.335} C_VEL
LIN {X 0,Y 578.657,Z 1140.753,A -85,B 0,C 180,E1 2055.227,E2 2055.227} C_VEL
LIN {X 0,Y 578.459,Z 1156.505,A -85,B 0,C 180,E1 2059.081,E2 2059.081} C_VEL
LIN {X 0,Y 578.404,Z 1166.332,A -85,B 0,C 180,E1 2062.48,E2 2062.48} C_VEL
LIN {X 0,Y 578.485,Z 1171.905,A -85,B 0,C 180,E1 2065.497,E2 2065.497} C_VEL
LIN {X 0,Y 578.489,Z 1174.657,A -85,B 0,C 180,E1 2068.501,E2 2068.501} C_VEL
LIN {X 0,Y 578.371,Z 1173.627,A -85,B 0,C 180,E1 2073.002,E2 2073.002} C_VEL
LIN {X 0,Y 578.512,Z 1167.914,A -85,B 0,C 180,E1 2076.765,E2 2076.765} C_VEL
LIN {X 0,Y 578.55,Z 1156.468,A -85,B 0,C 180,E1 2080.928,E2 2080.928} C_VEL
LIN {X 0,Y 578.742,Z 1140.609,A -85,B 0,C 180,E1 2084.801,E2 2084.801} C_VEL
LIN {X 0,Y 579.091,Z 1117.899,A -85,B 0,C 180,E1 2088.847,E2 2088.847} C_VEL
LIN {X 0,Y 579.792,Z 1089.976,A -85,B 0,C 180,E1 2092.621,E2 2092.621} C_VEL
LIN {X 0,Y 580.68,Z 1057.124,A -85,B 0,C 180,E1 2096.056,E2 2096.056} C_VEL
LIN {X 0,Y 581.728,Z 1021.454,A -85,B 0,C 180,E1 2098.948,E2 2098.948} C_VEL
LIN {X 0,Y 582.867,Z 981.985,A -85,B 0,C 180,E1 2101.368,E2 2101.368} C_VEL
LIN {X 0,Y 583.865,Z 941.929,A -85,B 0,C 180,E1 2103.129,E2 2103.129} C_VEL
LIN {X 0,Y 584.435,Z 904.3,A -85,B 0,C 180,E1 2104.223,E2 2104.223} C_VEL
LIN {X 0,Y 584.028,Z 856.427,A -85,B 0,C 180,E1 2105.062,E2 2105.062} C_VEL
LIN {X 0,Y 578.203,Z 843.44,A -85,B 0,C 180,E1 2105.737,E2 2105.737} C_VEL
LIN {X 0,Y 577.94,Z 843.44,A -85,B 0,C 180,E1 2110.918,E2 2110.918} C_VEL
LIN {X 0,Y 577.862,Z 843.44,A -85,B 0,C 180,E1 2117.196,E2 2117.196} C_VEL
LIN {X 0,Y 578.012,Z 843.44,A -85,B 0,C 180,E1 2122.956,E2 2122.956} C_VEL
LIN {X 0,Y 577.998,Z 843.44,A -85,B 0,C 180,E1 2128.408,E2 2128.408} C_VEL
LIN {X 0,Y 577.94,Z 843.44,A -85,B 0,C 180,E1 2133.555,E2 2133.555} C_VEL
LIN {X 0,Y 577.863,Z 843.44,A -85,B 0,C 180,E1 2138.482,E2 2138.482} C_VEL
LIN {X 0,Y 577.506,Z 843.44,A -85,B 0,C 180,E1 2141.664,E2 2141.664} C_VEL
LIN {X 0,Y 580.246,Z 859.645,A -85,B 0,C 180,E1 2141.975,E2 2141.975} C_VEL
LIN {X 0,Y 580.08,Z 894.05,A -85,B 0,C 180,E1 2142.628,E2 2142.628} C_VEL
LIN {X 0,Y 579.812,Z 924.073,A -85,B 0,C 180,E1 2143.795,E2 2143.795} C_VEL
LIN {X 0,Y 579.354,Z 951.664,A -85,B 0,C 180,E1 2145.493,E2 2145.493} C_VEL
LIN {X 0,Y 579.014,Z 976.606,A -85,B 0,C 180,E1 2147.734,E2 2147.734} C_VEL
LIN {X 0,Y 578.741,Z 997.092,A -85,B 0,C 180,E1 2150.4,E2 2150.4} C_VEL
LIN {X 0,Y 578.593,Z 1012.023,A -85,B 0,C 180,E1 2153.313,E2 2153.313} C_VEL
LIN {X 0,Y 578.546,Z 1021.033,A -85,B 0,C 180,E1 2156.248,E2 2156.248} C_VEL
LIN {X 0,Y 578.484,Z 1024.39,A -85,B 0,C 180,E1 2158.5,E2 2158.5} C_VEL
LIN {X 0,Y 578.479,Z 1024.315,A -85,B 0,C 180,E1 2161.499,E2 2161.499} C_VEL
LIN {X 0,Y 578.525,Z 1019.017,A -85,B 0,C 180,E1 2164.502,E2 2164.502} C_VEL
LIN {X 0,Y 578.605,Z 1008.019,A -85,B 0,C 180,E1 2167.517,E2 2167.517} C_VEL
LIN {X 0,Y 578.815,Z 991.4,A -85,B 0,C 180,E1 2170.359,E2 2170.359} C_VEL
LIN {X 0,Y 579.078,Z 970.177,A -85,B 0,C 180,E1 2172.839,E2 2172.839} C_VEL
LIN {X 0,Y 579.522,Z 943.859,A -85,B 0,C 180,E1 2174.971,E2 2174.971} C_VEL
LIN {X 0,Y 579.961,Z 914.888,A -85,B 0,C 180,E1 2176.54,E2 2176.54} C_VEL
LIN {X 0,Y 580.173,Z 883.824,A -85,B 0,C 180,E1 2177.545,E2 2177.545} C_VEL
LIN {X 0,Y 579.345,Z 848.286,A -85,B 0,C 180,E1 2178.109,E2 2178.109} C_VEL
LIN {X 0,Y 578.152,Z 843.44,A -85,B 0,C 180,E1 2178.247,E2 2178.247} C_VEL
LIN {X 0,Y 577.979,Z 843.44,A -85,B 0,C 180,E1 2183.522,E2 2183.522} C_VEL
LIN {X 0,Y 577.971,Z 843.44,A -85,B 0,C 180,E1 2188.13,E2 2188.13} C_VEL
LIN {X 0,Y 578.108,Z 843.44,A -85,B 0,C 180,E1 2193.362,E2 2193.362} C_VEL
LIN {X 0,Y 577.932,Z 843.44,A -85,B 0,C 180,E1 2198.953,E2 2198.953} C_VEL
LIN {X 0,Y 577.706,Z 843.44,A -85,B 0,C 180,E1 2204.955,E2 2204.955} C_VEL
LIN {X 0,Y 577.951,Z 843.44,A -85,B 0,C 180,E1 2209.433,E2 2209.433} C_VEL
LIN {X 0,Y 578.128,Z 843.44,A -85,B 0,C 180,E1 2214.816,E2 2214.816} C_VEL
LIN {X 0,Y 578.206,Z 843.44,A -85,B 0,C 180,E1 2218.745,E2 2218.745} C_VEL
LIN {X 0,Y 582.699,Z 854.827,A -85,B 0,C 180,E1 2219.203,E2 2219.203} C_VEL
LIN {X 0,Y 583.021,Z 912.863,A -85,B 0,C 180,E1 2220.194,E2 2220.194} C_VEL
LIN {X 0,Y 582.37,Z 953.031,A -85,B 0,C 180,E1 2221.507,E2 2221.507} C_VEL
LIN {X 0,Y 581.578,Z 989.984,A -85,B 0,C 180,E1 2223.342,E2 2223.342} C_VEL
LIN {X 0,Y 580.669,Z 1024.957,A -85,B 0,C 180,E1 2225.734,E2 2225.734} C_VEL
LIN {X 0,Y 579.794,Z 1056.149,A -85,B 0,C 180,E1 2228.554,E2 2228.554} C_VEL
LIN {X 0,Y 579.22,Z 1083.056,A -85,B 0,C 180,E1 2231.717,E2 2231.717} C_VEL
LIN {X 0,Y 578.777,Z 1105.862,A -85,B 0,C 180,E1 2235.23,E2 2235.23} C_VEL
LIN {X 0,Y 578.573,Z 1124.018,A -85,B 0,C 180,E1 2239.055,E2 2239.055} C_VEL
LIN {X 0,Y 578.484,Z 1136.284,A -85,B 0,C 180,E1 2242.895,E2 2242.895} C_VEL
LIN {X 0,Y 578.349,Z 1141.503,A -85,B 0,C 180,E1 2245.495,E2 2245.495} C_VEL
LIN {X 0,Y 578.346,Z 1144.613,A -85,B 0,C 180,E1 2248.499,E2 2248.499} C_VEL
LIN {X 0,Y 578.476,Z 1144.552,A -85,B 0,C 180,E1 2251.499,E2 2251.499} C_VEL
LIN {X 0,Y 578.534,Z 1140.206,A -85,B 0,C 180,E1 2255.221,E2 2255.221} C_VEL
LIN {X 0,Y 578.557,Z 1130.574,A -85,B 0,C 180,E1 2259.034,E2 2259.034} C_VEL
LIN {X 0,Y 578.705,Z 1115.377,A -85,B 0,C 180,E1 2262.849,E2 2262.849} C_VEL
LIN {X 0,Y 578.996,Z 1093.478,A -85,B 0,C 180,E1 2266.717,E2 2266.717} C_VEL
LIN {X 0,Y 579.567,Z 1068.283,A -85,B 0,C 180,E1 2270.032,E2 2270.032} C_VEL
LIN {X 0,Y 580.264,Z 1038.518,A -85,B 0,C 180,E1 2273.041,E2 2273.041} C_VEL
LIN {X 0,Y 581.159,Z 1004.924,A -85,B 0,C 180,E1 2275.631,E2 2275.631} C_VEL
LIN {X 0,Y 582.056,Z 968.871,A -85,B 0,C 180,E1 2277.692,E2 2277.692} C_VEL
LIN {X 0,Y 582.767,Z 931.893,A -85,B 0,C 180,E1 2279.172,E2 2279.172} C_VEL
LIN {X 0,Y 583.188,Z 894.076,A -85,B 0,C 180,E1 2280.106,E2 2280.106} C_VEL
LIN {X 0,Y 582.702,Z 854.775,A -85,B 0,C 180,E1 2280.708,E2 2280.708} C_VEL
LIN {X 0,Y 578.069,Z 843.44,A -85,B 0,C 180,E1 2281.19,E2 2281.19} C_VEL
LIN {X 0,Y 578.051,Z 843.44,A -85,B 0,C 180,E1 2287.045,E2 2287.045} C_VEL
LIN {X 0,Y 577.876,Z 843.44,A -85,B 0,C 180,E1 2292.94,E2 2292.94} C_VEL
LIN {X 0,Y 577.979,Z 843.44,A -85,B 0,C 180,E1 2297.181,E2 2297.181} C_VEL
LIN {X 0,Y 577.93,Z 843.44,A -85,B 0,C 180,E1 2302.951,E2 2302.951} C_VEL
LIN {X 0,Y 577.911,Z 843.44,A -85,B 0,C 180,E1 2308.404,E2 2308.404} C_VEL
LIN {X 0,Y 578.016,Z 843.44,A -85,B 0,C 180,E1 2313.561,E2 2313.561} C_VEL
LIN {X 0,Y 578.092,Z 843.44,A -85,B 0,C 180,E1 2318.492,E2 2318.492} C_VEL
LIN {X 0,Y 578.162,Z 843.44,A -85,B 0,C 180,E1 2323.26,E2 2323.26} C_VEL
LIN {X 0,Y 578.197,Z 843.44,A -85,B 0,C 180,E1 2327.909,E2 2327.909} C_VEL
LIN {X 0,Y 578.223,Z 843.44,A -85,B 0,C 180,E1 2332.478,E2 2332.478} C_VEL
LIN {X 0,Y 578.32,Z 843.44,A -85,B 0,C 180,E1 2337,E2 2337} C_VEL
LIN {X 0,Y 578.434,Z 843.44,A -85,B 0,C 180,E1 2341.5,E2 2341.5} C_VEL
LIN {X 0,Y 578.415,Z 843.44,A -85,B 0,C 180,E1 2346.01,E2 2346.01} C_VEL
LIN {X 0,Y 578.081,Z 843.44,A -85,B 0,C 180,E1 2347.599,E2 2347.599} C_VEL
LIN {X 0,Y 574.194,Z 843.44,A -85,B 0,C 180,E1 2349.291,E2 2349.291} C_VEL
LIN {X 0,Y 570.26,Z 843.44,A -85,B 0,C 180,E1 2351.006,E2 2351.006} C_VEL
LIN {X 0,Y 570.117,Z 843.44,A -85,B 0,C 180,E1 2357.043,E2 2357.043} C_VEL
LIN {X 0,Y 570.141,Z 843.44,A -85,B 0,C 180,E1 2361.825,E2 2361.825} C_VEL
LIN {X 0,Y 570.086,Z 843.44,A -85,B 0,C 180,E1 2366.838,E2 2366.838} C_VEL
LIN {X 0,Y 569.952,Z 843.44,A -85,B 0,C 180,E1 2372.091,E2 2372.091} C_VEL
LIN {X 0,Y 570.061,Z 843.44,A -85,B 0,C 180,E1 2377.65,E2 2377.65} C_VEL
LIN {X 0,Y 569.98,Z 843.44,A -85,B 0,C 180,E1 2383.678,E2 2383.678} C_VEL
LIN {X 0,Y 569.883,Z 843.44,A -85,B 0,C 180,E1 2388.378,E2 2388.378} C_VEL
LIN {X 0,Y 569.946,Z 844.176,A -85,B 0,C 180,E1 2393.751,E2 2393.751} C_VEL
LIN {X 0,Y 578.118,Z 861.143,A -85,B 0,C 180,E1 2394.597,E2 2394.597} C_VEL
LIN {X 0,Y 577.709,Z 912.731,A -85,B 0,C 180,E1 2395.529,E2 2395.529} C_VEL
LIN {X 0,Y 576.842,Z 953.669,A -85,B 0,C 180,E1 2396.889,E2 2396.889} C_VEL
LIN {X 0,Y 575.639,Z 992.192,A -85,B 0,C 180,E1 2398.781,E2 2398.781} C_VEL
LIN {X 0,Y 574.34,Z 1028.492,A -85,B 0,C 180,E1 2401.181,E2 2401.181} C_VEL
LIN {X 0,Y 573.075,Z 1062.349,A -85,B 0,C 180,E1 2404.081,E2 2404.081} C_VEL
LIN {X 0,Y 572.005,Z 1093.564,A -85,B 0,C 180,E1 2407.507,E2 2407.507} C_VEL
LIN {X 0,Y 571.272,Z 1119.243,A -85,B 0,C 180,E1 2411.106,E2 2411.106} C_VEL
LIN {X 0,Y 570.821,Z 1140.438,A -85,B 0,C 180,E1 2414.954,E2 2414.954} C_VEL
LIN {X 0,Y 570.6,Z 1156.843,A -85,B 0,C 180,E1 2419.026,E2 2419.026} C_VEL
LIN {X 0,Y 570.521,Z 1166.332,A -85,B 0,C 180,E1 2422.375,E2 2422.375} C_VEL
LIN {X 0,Y 570.612,Z 1171.905,A -85,B 0,C 180,E1 2425.435,E2 2425.435} C_VEL
LIN {X 0,Y 570.589,Z 1174.657,A -85,B 0,C 180,E1 2428.48,E2 2428.48} C_VEL
LIN {X 0,Y 570.465,Z 1173.627,A -85,B 0,C 180,E1 2433.044,E2 2433.044} C_VEL
LIN {X 0,Y 570.605,Z 1167.915,A -85,B 0,C 180,E1 2436.859,E2 2436.859} C_VEL
LIN {X 0,Y 570.654,Z 1156.743,A -85,B 0,C 180,E1 2441.002,E2 2441.002} C_VEL
LIN {X 0,Y 570.921,Z 1140.308,A -85,B 0,C 180,E1 2445.069,E2 2445.069} C_VEL
LIN {X 0,Y 571.346,Z 1117.109,A -85,B 0,C 180,E1 2449.234,E2 2449.234} C_VEL
LIN {X 0,Y 572.197,Z 1089.16,A -85,B 0,C 180,E1 2453.034,E2 2453.034} C_VEL
LIN {X 0,Y 573.323,Z 1056.353,A -85,B 0,C 180,E1 2456.487,E2 2456.487} C_VEL
LIN {X 0,Y 574.642,Z 1020.29,A -85,B 0,C 180,E1 2459.423,E2 2459.423} C_VEL
LIN {X 0,Y 575.963,Z 981.896,A -85,B 0,C 180,E1 2461.792,E2 2461.792} C_VEL
LIN {X 0,Y 577.219,Z 940.819,A -85,B 0,C 180,E1 2463.605,E2 2463.605} C_VEL
LIN {X 0,Y 577.935,Z 902.792,A -85,B 0,C 180,E1 2464.697,E2 2464.697} C_VEL
LIN {X 0,Y 577.71,Z 859.523,A -85,B 0,C 180,E1 2465.456,E2 2465.456} C_VEL
LIN {X 0,Y 570.203,Z 843.44,A -85,B 0,C 180,E1 2466.266,E2 2466.266} C_VEL
LIN {X 0,Y 569.915,Z 843.44,A -85,B 0,C 180,E1 2471.943,E2 2471.943} C_VEL
LIN {X 0,Y 569.94,Z 843.44,A -85,B 0,C 180,E1 2478.387,E2 2478.387} C_VEL
LIN {X 0,Y 570.17,Z 843.44,A -85,B 0,C 180,E1 2484.256,E2 2484.256} C_VEL
LIN {X 0,Y 570.106,Z 843.44,A -85,B 0,C 180,E1 2489.697,E2 2489.697} C_VEL
LIN {X 0,Y 570.009,Z 843.44,A -85,B 0,C 180,E1 2494.851,E2 2494.851} C_VEL
LIN {X 0,Y 569.901,Z 843.44,A -85,B 0,C 180,E1 2499.796,E2 2499.796} C_VEL
LIN {X 0,Y 569.657,Z 843.44,A -85,B 0,C 180,E1 2501.402,E2 2501.402} C_VEL
LIN {X 0,Y 572.747,Z 861.107,A -85,B 0,C 180,E1 2501.751,E2 2501.751} C_VEL
LIN {X 0,Y 572.55,Z 894.246,A -85,B 0,C 180,E1 2502.399,E2 2502.399} C_VEL
LIN {X 0,Y 572.194,Z 924.066,A -85,B 0,C 180,E1 2503.573,E2 2503.573} C_VEL
LIN {X 0,Y 571.63,Z 951.937,A -85,B 0,C 180,E1 2505.315,E2 2505.315} C_VEL
LIN {X 0,Y 571.223,Z 976.603,A -85,B 0,C 180,E1 2507.564,E2 2507.564} C_VEL
LIN {X 0,Y 570.889,Z 997.091,A -85,B 0,C 180,E1 2510.266,E2 2510.266} C_VEL
LIN {X 0,Y 570.704,Z 1011.717,A -85,B 0,C 180,E1 2513.143,E2 2513.143} C_VEL
LIN {X 0,Y 570.645,Z 1021.033,A -85,B 0,C 180,E1 2516.196,E2 2516.196} C_VEL
LIN {X 0,Y 570.593,Z 1024.391,A -85,B 0,C 180,E1 2518.479,E2 2518.479} C_VEL
LIN {X 0,Y 570.588,Z 1024.314,A -85,B 0,C 180,E1 2521.52,E2 2521.52} C_VEL
LIN {X 0,Y 570.652,Z 1019.019,A -85,B 0,C 180,E1 2524.564,E2 2524.564} C_VEL
LIN {X 0,Y 570.72,Z 1008.023,A -85,B 0,C 180,E1 2527.621,E2 2527.621} C_VEL
LIN {X 0,Y 570.985,Z 991.407,A -85,B 0,C 180,E1 2530.502,E2 2530.502} C_VEL
LIN {X 0,Y 571.311,Z 970.186,A -85,B 0,C 180,E1 2533.017,E2 2533.017} C_VEL
LIN {X 0,Y 571.857,Z 943.865,A -85,B 0,C 180,E1 2535.176,E2 2535.176} C_VEL
LIN {X 0,Y 572.36,Z 914.901,A -85,B 0,C 180,E1 2536.766,E2 2536.766} C_VEL
LIN {X 0,Y 572.636,Z 885.344,A -85,B 0,C 180,E1 2537.749,E2 2537.749} C_VEL
LIN {X 0,Y 571.925,Z 849.98,A -85,B 0,C 180,E1 2538.331,E2 2538.331} C_VEL
LIN {X 0,Y 570.193,Z 843.44,A -85,B 0,C 180,E1 2538.498,E2 2538.498} C_VEL
LIN {X 0,Y 570.103,Z 843.44,A -85,B 0,C 180,E1 2543.473,E2 2543.473} C_VEL
LIN {X 0,Y 569.999,Z 843.44,A -85,B 0,C 180,E1 2548.763,E2 2548.763} C_VEL
LIN {X 0,Y 570.121,Z 843.44,A -85,B 0,C 180,E1 2554.582,E2 2554.582} C_VEL
LIN {X 0,Y 569.987,Z 843.44,A -85,B 0,C 180,E1 2559.612,E2 2559.612} C_VEL
LIN {X 0,Y 569.785,Z 843.44,A -85,B 0,C 180,E1 2565.839,E2 2565.839} C_VEL
LIN {X 0,Y 570.023,Z 843.44,A -85,B 0,C 180,E1 2570.393,E2 2570.393} C_VEL
LIN {X 0,Y 570.236,Z 843.44,A -85,B 0,C 180,E1 2576.109,E2 2576.109} C_VEL
LIN {X 0,Y 570.281,Z 843.44,A -85,B 0,C 180,E1 2578.288,E2 2578.288} C_VEL
LIN {X 0,Y 576.023,Z 859.514,A -85,B 0,C 180,E1 2578.874,E2 2578.874} C_VEL
LIN {X 0,Y 576.126,Z 913.83,A -85,B 0,C 180,E1 2579.828,E2 2579.828} C_VEL
LIN {X 0,Y 575.352,Z 953.228,A -85,B 0,C 180,E1 2581.136,E2 2581.136} C_VEL
LIN {X 0,Y 574.339,Z 990.907,A -85,B 0,C 180,E1 2583.037,E2 2583.037} C_VEL
LIN {X 0,Y 573.246,Z 1025.632,A -85,B 0,C 180,E1 2585.456,E2 2585.456} C_VEL
LIN {X 0,Y 572.229,Z 1056.143,A -85,B 0,C 180,E1 2588.256,E2 2588.256} C_VEL
LIN {X 0,Y 571.505,Z 1083.052,A -85,B 0,C 180,E1 2591.462,E2 2591.462} C_VEL
LIN {X 0,Y 570.976,Z 1105.656,A -85,B 0,C 180,E1 2594.987,E2 2594.987} C_VEL
LIN {X 0,Y 570.647,Z 1122.414,A -85,B 0,C 180,E1 2598.499,E2 2598.499} C_VEL
LIN {X 0,Y 570.546,Z 1135.224,A -85,B 0,C 180,E1 2602.374,E2 2602.374} C_VEL
LIN {X 0,Y 570.478,Z 1141.503,A -85,B 0,C 180,E1 2605.432,E2 2605.432} C_VEL
LIN {X 0,Y 570.457,Z 1144.613,A -85,B 0,C 180,E1 2608.478,E2 2608.478} C_VEL
LIN {X 0,Y 570.577,Z 1144.553,A -85,B 0,C 180,E1 2611.52,E2 2611.52} C_VEL
LIN {X 0,Y 570.648,Z 1140.399,A -85,B 0,C 180,E1 2615.176,E2 2615.176} C_VEL
LIN {X 0,Y 570.665,Z 1130.576,A -85,B 0,C 180,E1 2619.16,E2 2619.16} C_VEL
LIN {X 0,Y 570.866,Z 1115.38,A -85,B 0,C 180,E1 2623.029,E2 2623.029} C_VEL
LIN {X 0,Y 571.237,Z 1093.48,A -85,B 0,C 180,E1 2626.951,E2 2626.951} C_VEL
LIN {X 0,Y 571.91,Z 1068.109,A -85,B 0,C 180,E1 2630.333,E2 2630.333} C_VEL
LIN {X 0,Y 572.814,Z 1038.527,A -85,B 0,C 180,E1 2633.359,E2 2633.359} C_VEL
LIN {X 0,Y 573.886,Z 1005.216,A -85,B 0,C 180,E1 2635.961,E2 2635.961} C_VEL
LIN {X 0,Y 574.911,Z 970.414,A -85,B 0,C 180,E1 2637.989,E2 2637.989} C_VEL
LIN {X 0,Y 575.793,Z 933.003,A -85,B 0,C 180,E1 2639.525,E2 2639.525} C_VEL
LIN {X 0,Y 576.366,Z 893.769,A -85,B 0,C 180,E1 2640.505,E2 2640.505} C_VEL
LIN {X 0,Y 575.88,Z 857.03,A -85,B 0,C 180,E1 2641.08,E2 2641.08} C_VEL
LIN {X 0,Y 570.063,Z 843.44,A -85,B 0,C 180,E1 2641.696,E2 2641.696} C_VEL
LIN {X 0,Y 570.141,Z 843.44,A -85,B 0,C 180,E1 2647.648,E2 2647.648} C_VEL
LIN {X 0,Y 569.933,Z 843.44,A -85,B 0,C 180,E1 2654.176,E2 2654.176} C_VEL
LIN {X 0,Y 569.98,Z 843.44,A -85,B 0,C 180,E1 2658.393,E2 2658.393} C_VEL
LIN {X 0,Y 569.975,Z 843.44,A -85,B 0,C 180,E1 2664.244,E2 2664.244} C_VEL
LIN {X 0,Y 570.032,Z 843.44,A -85,B 0,C 180,E1 2669.695,E2 2669.695} C_VEL
LIN {X 0,Y 570.156,Z 843.44,A -85,B 0,C 180,E1 2674.86,E2 2674.86} C_VEL
LIN {X 0,Y 570.249,Z 843.44,A -85,B 0,C 180,E1 2679.811,E2 2679.811} C_VEL
LIN {X 0,Y 570.405,Z 843.44,A -85,B 0,C 180,E1 2686.181,E2 2686.181} C_VEL
LIN {X 0,Y 570.314,Z 843.44,A -85,B 0,C 180,E1 2692.373,E2 2692.373} C_VEL
LIN {X 0,Y 570.412,Z 843.44,A -85,B 0,C 180,E1 2696.958,E2 2696.958} C_VEL
LIN {X 0,Y 570.536,Z 843.44,A -85,B 0,C 180,E1 2701.521,E2 2701.521} C_VEL
LIN {X 0,Y 570.483,Z 843.44,A -85,B 0,C 180,E1 2706.094,E2 2706.094} C_VEL
LIN {X 0,Y 570.26,Z 843.44,A -85,B 0,C 180,E1 2711.006,E2 2711.006} C_VEL
LIN {X 0,Y 566.197,Z 843.44,A -85,B 0,C 180,E1 2712.717,E2 2712.717} C_VEL
LIN {X 0,Y 562.22,Z 843.44,A -85,B 0,C 180,E1 2714.453,E2 2714.453} C_VEL
LIN {X 0,Y 562.258,Z 843.44,A -85,B 0,C 180,E1 2720.49,E2 2720.49} C_VEL
LIN {X 0,Y 562.275,Z 843.44,A -85,B 0,C 180,E1 2725.519,E2 2725.519} C_VEL
LIN {X 0,Y 562.079,Z 843.44,A -85,B 0,C 180,E1 2730.782,E2 2730.782} C_VEL
LIN {X 0,Y 562.114,Z 843.44,A -85,B 0,C 180,E1 2736.337,E2 2736.337} C_VEL
LIN {X 0,Y 562.045,Z 843.44,A -85,B 0,C 180,E1 2742.332,E2 2742.332} C_VEL
LIN {X 0,Y 561.962,Z 843.44,A -85,B 0,C 180,E1 2747.656,E2 2747.656} C_VEL
LIN {X 0,Y 562.023,Z 843.44,A -85,B 0,C 180,E1 2753.121,E2 2753.121} C_VEL
LIN {X 0,Y 571.351,Z 862.897,A -85,B 0,C 180,E1 2754.14,E2 2754.14} C_VEL
LIN {X 0,Y 571.164,Z 913.112,A -85,B 0,C 180,E1 2755.088,E2 2755.088} C_VEL
LIN {X 0,Y 570.129,Z 953.179,A -85,B 0,C 180,E1 2756.428,E2 2756.428} C_VEL
LIN {X 0,Y 568.789,Z 990.406,A -85,B 0,C 180,E1 2758.255,E2 2758.255} C_VEL
LIN {X 0,Y 567.296,Z 1026.025,A -85,B 0,C 180,E1 2760.593,E2 2760.593} C_VEL
LIN {X 0,Y 565.772,Z 1060.554,A -85,B 0,C 180,E1 2763.538,E2 2763.538} C_VEL
LIN {X 0,Y 564.551,Z 1091.35,A -85,B 0,C 180,E1 2766.907,E2 2766.907} C_VEL
LIN {X 0,Y 563.566,Z 1117.899,A -85,B 0,C 180,E1 2770.613,E2 2770.613} C_VEL
LIN {X 0,Y 563.007,Z 1140.303,A -85,B 0,C 180,E1 2774.713,E2 2774.713} C_VEL
LIN {X 0,Y 562.713,Z 1156.844,A -85,B 0,C 180,E1 2778.87,E2 2778.87} C_VEL
LIN {X 0,Y 562.661,Z 1166.332,A -85,B 0,C 180,E1 2782.268,E2 2782.268} C_VEL
LIN {X 0,Y 562.717,Z 1171.905,A -85,B 0,C 180,E1 2785.371,E2 2785.371} C_VEL
LIN {X 0,Y 562.683,Z 1174.657,A -85,B 0,C 180,E1 2788.459,E2 2788.459} C_VEL
LIN {X 0,Y 562.561,Z 1173.627,A -85,B 0,C 180,E1 2793.086,E2 2793.086} C_VEL
LIN {X 0,Y 562.727,Z 1167.915,A -85,B 0,C 180,E1 2796.955,E2 2796.955} C_VEL
LIN {X 0,Y 562.752,Z 1156.744,A -85,B 0,C 180,E1 2801.159,E2 2801.159} C_VEL
LIN {X 0,Y 563.081,Z 1140.229,A -85,B 0,C 180,E1 2805.3,E2 2805.3} C_VEL
LIN {X 0,Y 563.595,Z 1117.913,A -85,B 0,C 180,E1 2809.384,E2 2809.384} C_VEL
LIN {X 0,Y 564.634,Z 1089.666,A -85,B 0,C 180,E1 2813.3,E2 2813.3} C_VEL
LIN {X 0,Y 565.935,Z 1057.383,A -85,B 0,C 180,E1 2816.764,E2 2816.764} C_VEL
LIN {X 0,Y 567.494,Z 1022.248,A -85,B 0,C 180,E1 2819.689,E2 2819.689} C_VEL
LIN {X 0,Y 569.11,Z 982.215,A -85,B 0,C 180,E1 2822.204,E2 2822.204} C_VEL
LIN {X 0,Y 570.519,Z 941.945,A -85,B 0,C 180,E1 2824.007,E2 2824.007} C_VEL
LIN {X 0,Y 571.444,Z 902.691,A -85,B 0,C 180,E1 2825.151,E2 2825.151} C_VEL
LIN {X 0,Y 571.072,Z 861.922,A -85,B 0,C 180,E1 2825.895,E2 2825.895} C_VEL
LIN {X 0,Y 562.246,Z 843.44,A -85,B 0,C 180,E1 2826.874,E2 2826.874} C_VEL
LIN {X 0,Y 561.959,Z 843.44,A -85,B 0,C 180,E1 2832.346,E2 2832.346} C_VEL
LIN {X 0,Y 561.966,Z 843.44,A -85,B 0,C 180,E1 2837.661,E2 2837.661} C_VEL
LIN {X 0,Y 562.225,Z 843.44,A -85,B 0,C 180,E1 2843.896,E2 2843.896} C_VEL
LIN {X 0,Y 562.196,Z 843.44,A -85,B 0,C 180,E1 2849.525,E2 2849.525} C_VEL
LIN {X 0,Y 562.097,Z 843.44,A -85,B 0,C 180,E1 2854.472,E2 2854.472} C_VEL
LIN {X 0,Y 562.006,Z 843.44,A -85,B 0,C 180,E1 2859.5,E2 2859.5} C_VEL
LIN {X 0,Y 561.768,Z 843.44,A -85,B 0,C 180,E1 2861.131,E2 2861.131} C_VEL
LIN {X 0,Y 565.23,Z 860.506,A -85,B 0,C 180,E1 2861.492,E2 2861.492} C_VEL
LIN {X 0,Y 565.014,Z 893.172,A -85,B 0,C 180,E1 2862.124,E2 2862.124} C_VEL
LIN {X 0,Y 564.565,Z 924.059,A -85,B 0,C 180,E1 2863.345,E2 2863.345} C_VEL
LIN {X 0,Y 563.903,Z 952.567,A -85,B 0,C 180,E1 2865.16,E2 2865.16} C_VEL
LIN {X 0,Y 563.421,Z 976.601,A -85,B 0,C 180,E1 2867.389,E2 2867.389} C_VEL
LIN {X 0,Y 563.054,Z 997.09,A -85,B 0,C 180,E1 2870.129,E2 2870.129} C_VEL
LIN {X 0,Y 562.833,Z 1011.716,A -85,B 0,C 180,E1 2873.047,E2 2873.047} C_VEL
LIN {X 0,Y 562.757,Z 1021.032,A -85,B 0,C 180,E1 2876.143,E2 2876.143} C_VEL
LIN {X 0,Y 562.691,Z 1024.391,A -85,B 0,C 180,E1 2878.458,E2 2878.458} C_VEL
LIN {X 0,Y 562.686,Z 1024.313,A -85,B 0,C 180,E1 2881.541,E2 2881.541} C_VEL
LIN {X 0,Y 562.754,Z 1019.022,A -85,B 0,C 180,E1 2884.628,E2 2884.628} C_VEL
LIN {X 0,Y 562.846,Z 1008.026,A -85,B 0,C 180,E1 2887.728,E2 2887.728} C_VEL
LIN {X 0,Y 563.151,Z 991.413,A -85,B 0,C 180,E1 2890.65,E2 2890.65} C_VEL
LIN {X 0,Y 563.535,Z 970.193,A -85,B 0,C 180,E1 2893.199,E2 2893.199} C_VEL
LIN {X 0,Y 564.163,Z 944.796,A -85,B 0,C 180,E1 2895.325,E2 2895.325} C_VEL
LIN {X 0,Y 564.766,Z 916.021,A -85,B 0,C 180,E1 2896.948,E2 2896.948} C_VEL
LIN {X 0,Y 565.112,Z 885.346,A -85,B 0,C 180,E1 2897.994,E2 2897.994} C_VEL
LIN {X 0,Y 564.516,Z 851.894,A -85,B 0,C 180,E1 2898.556,E2 2898.556} C_VEL
LIN {X 0,Y 562.216,Z 843.44,A -85,B 0,C 180,E1 2898.757,E2 2898.757} C_VEL
LIN {X 0,Y 562.159,Z 843.44,A -85,B 0,C 180,E1 2903.825,E2 2903.825} C_VEL
LIN {X 0,Y 562.069,Z 843.44,A -85,B 0,C 180,E1 2909.001,E2 2909.001} C_VEL
LIN {X 0,Y 562.243,Z 843.44,A -85,B 0,C 180,E1 2914.434,E2 2914.434} C_VEL
LIN {X 0,Y 562.012,Z 843.44,A -85,B 0,C 180,E1 2920.278,E2 2920.278} C_VEL
LIN {X 0,Y 561.902,Z 843.44,A -85,B 0,C 180,E1 2926.673,E2 2926.673} C_VEL
LIN {X 0,Y 562.107,Z 843.44,A -85,B 0,C 180,E1 2931.716,E2 2931.716} C_VEL
LIN {X 0,Y 562.281,Z 843.44,A -85,B 0,C 180,E1 2937.413,E2 2937.413} C_VEL
LIN {X 0,Y 562.369,Z 844.04,A -85,B 0,C 180,E1 2937.803,E2 2937.803} C_VEL
LIN {X 0,Y 569.256,Z 860.597,A -85,B 0,C 180,E1 2938.478,E2 2938.478} C_VEL
LIN {X 0,Y 569.282,Z 914.08,A -85,B 0,C 180,E1 2939.434,E2 2939.434} C_VEL
LIN {X 0,Y 568.429,Z 951.739,A -85,B 0,C 180,E1 2940.685,E2 2940.685} C_VEL
LIN {X 0,Y 567.228,Z 989.422,A -85,B 0,C 180,E1 2942.579,E2 2942.579} C_VEL
LIN {X 0,Y 565.869,Z 1024.772,A -85,B 0,C 180,E1 2945.043,E2 2945.043} C_VEL
LIN {X 0,Y 564.682,Z 1056.136,A -85,B 0,C 180,E1 2947.951,E2 2947.951} C_VEL
LIN {X 0,Y 563.797,Z 1083.048,A -85,B 0,C 180,E1 2951.199,E2 2951.199} C_VEL
LIN {X 0,Y 563.163,Z 1105.37,A -85,B 0,C 180,E1 2954.722,E2 2954.722} C_VEL
LIN {X 0,Y 562.768,Z 1122.498,A -85,B 0,C 180,E1 2958.358,E2 2958.358} C_VEL
LIN {X 0,Y 562.675,Z 1135.223,A -85,B 0,C 180,E1 2962.267,E2 2962.267} C_VEL
LIN {X 0,Y 562.577,Z 1141.502,A -85,B 0,C 180,E1 2965.368,E2 2965.368} C_VEL
LIN {X 0,Y 562.555,Z 1144.612,A -85,B 0,C 180,E1 2968.457,E2 2968.457} C_VEL
LIN {X 0,Y 562.672,Z 1144.553,A -85,B 0,C 180,E1 2971.541,E2 2971.541} C_VEL
LIN {X 0,Y 562.7,Z 1140.043,A -85,B 0,C 180,E1 2975.456,E2 2975.456} C_VEL
LIN {X 0,Y 562.786,Z 1130.578,A -85,B 0,C 180,E1 2979.289,E2 2979.289} C_VEL
LIN {X 0,Y 563.002,Z 1115.384,A -85,B 0,C 180,E1 2983.214,E2 2983.214} C_VEL
LIN {X 0,Y 563.495,Z 1093.483,A -85,B 0,C 180,E1 2987.191,E2 2987.191} C_VEL
LIN {X 0,Y 564.26,Z 1068.114,A -85,B 0,C 180,E1 2990.621,E2 2990.621} C_VEL
LIN {X 0,Y 565.382,Z 1038.537,A -85,B 0,C 180,E1 2993.684,E2 2993.684} C_VEL
LIN {X 0,Y 566.661,Z 1004.599,A -85,B 0,C 180,E1 2996.362,E2 2996.362} C_VEL
LIN {X 0,Y 567.839,Z 970.223,A -85,B 0,C 180,E1 2998.38,E2 2998.38} C_VEL
LIN {X 0,Y 568.864,Z 933.545,A -85,B 0,C 180,E1 2999.903,E2 2999.903} C_VEL
LIN {X 0,Y 569.551,Z 894.947,A -85,B 0,C 180,E1 3000.891,E2 3000.891} C_VEL
LIN {X 0,Y 569.039,Z 859.549,A -85,B 0,C 180,E1 3001.461,E2 3001.461} C_VEL
LIN {X 0,Y 562.071,Z 843.44,A -85,B 0,C 180,E1 3002.208,E2 3002.208} C_VEL
LIN {X 0,Y 562.131,Z 843.44,A -85,B 0,C 180,E1 3008.28,E2 3008.28} C_VEL
LIN {X 0,Y 562.02,Z 843.44,A -85,B 0,C 180,E1 3014.463,E2 3014.463} C_VEL
LIN {X 0,Y 562.03,Z 843.44,A -85,B 0,C 180,E1 3019.724,E2 3019.724} C_VEL
LIN {X 0,Y 561.986,Z 843.44,A -85,B 0,C 180,E1 3025.548,E2 3025.548} C_VEL
LIN {X 0,Y 562.064,Z 843.44,A -85,B 0,C 180,E1 3030.999,E2 3030.999} C_VEL
LIN {X 0,Y 562.226,Z 843.44,A -85,B 0,C 180,E1 3036.297,E2 3036.297} C_VEL
LIN {X 0,Y 562.326,Z 843.44,A -85,B 0,C 180,E1 3041.152,E2 3041.152} C_VEL
LIN {X 0,Y 562.463,Z 843.44,A -85,B 0,C 180,E1 3045.982,E2 3045.982} C_VEL
LIN {X 0,Y 562.408,Z 843.44,A -85,B 0,C 180,E1 3052.266,E2 3052.266} C_VEL
LIN {X 0,Y 562.504,Z 843.44,A -85,B 0,C 180,E1 3056.915,E2 3056.915} C_VEL
LIN {X 0,Y 562.625,Z 843.44,A -85,B 0,C 180,E1 3061.543,E2 3061.543} C_VEL
LIN {X 0,Y 562.563,Z 843.44,A -85,B 0,C 180,E1 3066.18,E2 3066.18} C_VEL
LIN {X 0,Y 562.256,Z 843.44,A -85,B 0,C 180,E1 3072.44,E2 3072.44} C_VEL
LIN {X 0,Y 562.22,Z 843.44,A -85,B 0,C 180,E1 3074.453,E2 3074.453} C_VEL
LIN {X 0,Y 558.242,Z 843.44,A -85,B 0,C 180,E1 3076.195,E2 3076.195} C_VEL
LIN {X 0,Y 554.245,Z 843.44,A -85,B 0,C 180,E1 3077.962,E2 3077.962} C_VEL
LIN {X 0,Y 554.279,Z 843.44,A -85,B 0,C 180,E1 3082.483,E2 3082.483} C_VEL
LIN {X 0,Y 554.203,Z 843.44,A -85,B 0,C 180,E1 3087.672,E2 3087.672} C_VEL
LIN {X 0,Y 554.071,Z 843.44,A -85,B 0,C 180,E1 3093.127,E2 3093.127} C_VEL
LIN {X 0,Y 554.139,Z 843.44,A -85,B 0,C 180,E1 3098.931,E2 3098.931} C_VEL
LIN {X 0,Y 554.159,Z 843.44,A -85,B 0,C 180,E1 3104.734,E2 3104.734} C_VEL
LIN {X 0,Y 554.059,Z 843.44,A -85,B 0,C 180,E1 3111.058,E2 3111.058} C_VEL
LIN {X 0,Y 554.127,Z 843.44,A -85,B 0,C 180,E1 3112.528,E2 3112.528} C_VEL
LIN {X 0,Y 560.422,Z 857.28,A -85,B 0,C 180,E1 3113.24,E2 3113.24} C_VEL
LIN {X 0,Y 565.194,Z 866.354,A -85,B 0,C 180,E1 3113.741,E2 3113.741} C_VEL
LIN {X 0,Y 564.648,Z 913.129,A -85,B 0,C 180,E1 3114.626,E2 3114.626} C_VEL
LIN {X 0,Y 563.445,Z 953.912,A -85,B 0,C 180,E1 3116.006,E2 3116.006} C_VEL
LIN {X 0,Y 561.856,Z 992.076,A -85,B 0,C 180,E1 3117.918,E2 3117.918} C_VEL
LIN {X 0,Y 560.097,Z 1028.076,A -85,B 0,C 180,E1 3120.342,E2 3120.342} C_VEL
LIN {X 0,Y 558.314,Z 1062.886,A -85,B 0,C 180,E1 3123.398,E2 3123.398} C_VEL
LIN {X 0,Y 556.916,Z 1092.964,A -85,B 0,C 180,E1 3126.783,E2 3126.783} C_VEL
LIN {X 0,Y 555.788,Z 1119.837,A -85,B 0,C 180,E1 3130.659,E2 3130.659} C_VEL
LIN {X 0,Y 555.199,Z 1140.129,A -85,B 0,C 180,E1 3134.457,E2 3134.457} C_VEL
LIN {X 0,Y 554.848,Z 1156.438,A -85,B 0,C 180,E1 3138.59,E2 3138.59} C_VEL
LIN {X 0,Y 554.774,Z 1166.332,A -85,B 0,C 180,E1 3142.157,E2 3142.157} C_VEL
LIN {X 0,Y 554.819,Z 1171.905,A -85,B 0,C 180,E1 3145.305,E2 3145.305} C_VEL
LIN {X 0,Y 554.777,Z 1174.657,A -85,B 0,C 180,E1 3148.437,E2 3148.437} C_VEL
LIN {X 0,Y 554.672,Z 1173.627,A -85,B 0,C 180,E1 3153.13,E2 3153.13} C_VEL
LIN {X 0,Y 554.838,Z 1167.915,A -85,B 0,C 180,E1 3157.055,E2 3157.055} C_VEL
LIN {X 0,Y 554.888,Z 1157.772,A -85,B 0,C 180,E1 3161.012,E2 3161.012} C_VEL
LIN {X 0,Y 555.232,Z 1141.302,A -85,B 0,C 180,E1 3165.287,E2 3165.287} C_VEL
LIN {X 0,Y 555.869,Z 1118.336,A -85,B 0,C 180,E1 3169.593,E2 3169.593} C_VEL
LIN {X 0,Y 557.102,Z 1089.668,A -85,B 0,C 180,E1 3173.634,E2 3173.634} C_VEL
LIN {X 0,Y 558.631,Z 1057.244,A -85,B 0,C 180,E1 3177.156,E2 3177.156} C_VEL
LIN {X 0,Y 560.472,Z 1021.062,A -85,B 0,C 180,E1 3180.187,E2 3180.187} C_VEL
LIN {X 0,Y 562.288,Z 981.672,A -85,B 0,C 180,E1 3182.672,E2 3182.672} C_VEL
LIN {X 0,Y 563.969,Z 940.268,A -85,B 0,C 180,E1 3184.525,E2 3184.525} C_VEL
LIN {X 0,Y 565.022,Z 901.58,A -85,B 0,C 180,E1 3185.638,E2 3185.638} C_VEL
LIN {X 0,Y 564.82,Z 865.167,A -85,B 0,C 180,E1 3186.306,E2 3186.306} C_VEL
LIN {X 0,Y 554.351,Z 844.025,A -85,B 0,C 180,E1 3187.442,E2 3187.442} C_VEL
LIN {X 0,Y 554.015,Z 843.44,A -85,B 0,C 180,E1 3193.1,E2 3193.1} C_VEL
LIN {X 0,Y 554.108,Z 843.44,A -85,B 0,C 180,E1 3199.024,E2 3199.024} C_VEL
LIN {X 0,Y 554.308,Z 843.44,A -85,B 0,C 180,E1 3205.033,E2 3205.033} C_VEL
LIN {X 0,Y 554.314,Z 843.44,A -85,B 0,C 180,E1 3210.939,E2 3210.939} C_VEL
LIN {X 0,Y 554.163,Z 843.44,A -85,B 0,C 180,E1 3215.807,E2 3215.807} C_VEL
LIN {X 0,Y 553.915,Z 843.44,A -85,B 0,C 180,E1 3220.853,E2 3220.853} C_VEL
LIN {X 0,Y 557.749,Z 861.114,A -85,B 0,C 180,E1 3221.243,E2 3221.243} C_VEL
LIN {X 0,Y 557.472,Z 894.678,A -85,B 0,C 180,E1 3221.922,E2 3221.922} C_VEL
LIN {X 0,Y 556.955,Z 924.052,A -85,B 0,C 180,E1 3223.111,E2 3223.111} C_VEL
LIN {X 0,Y 556.235,Z 952.547,A -85,B 0,C 180,E1 3224.951,E2 3224.951} C_VEL
LIN {X 0,Y 555.624,Z 976.599,A -85,B 0,C 180,E1 3227.209,E2 3227.209} C_VEL
LIN {X 0,Y 555.197,Z 997.089,A -85,B 0,C 180,E1 3229.988,E2 3229.988} C_VEL
LIN {X 0,Y 554.956,Z 1011.716,A -85,B 0,C 180,E1 3232.948,E2 3232.948} C_VEL
LIN {X 0,Y 554.885,Z 1021.031,A -85,B 0,C 180,E1 3236.088,E2 3236.088} C_VEL
LIN {X 0,Y 554.789,Z 1024.391,A -85,B 0,C 180,E1 3238.436,E2 3238.436} C_VEL
LIN {X 0,Y 554.784,Z 1024.312,A -85,B 0,C 180,E1 3241.563,E2 3241.563} C_VEL
LIN {X 0,Y 554.86,Z 1019.025,A -85,B 0,C 180,E1 3244.694,E2 3244.694} C_VEL
LIN {X 0,Y 554.973,Z 1008.03,A -85,B 0,C 180,E1 3247.839,E2 3247.839} C_VEL
LIN {X 0,Y 555.289,Z 992.755,A -85,B 0,C 180,E1 3250.604,E2 3250.604} C_VEL
LIN {X 0,Y 555.735,Z 972.12,A -85,B 0,C 180,E1 3253.188,E2 3253.188} C_VEL
LIN {X 0,Y 556.469,Z 946.019,A -85,B 0,C 180,E1 3255.453,E2 3255.453} C_VEL
LIN {X 0,Y 557.174,Z 917.099,A -85,B 0,C 180,E1 3257.135,E2 3257.135} C_VEL
LIN {X 0,Y 557.591,Z 885.996,A -85,B 0,C 180,E1 3258.23,E2 3258.23} C_VEL
LIN {X 0,Y 557.055,Z 853.577,A -85,B 0,C 180,E1 3258.792,E2 3258.792} C_VEL
LIN {X 0,Y 554.267,Z 843.44,A -85,B 0,C 180,E1 3259.028,E2 3259.028} C_VEL
LIN {X 0,Y 554.2,Z 843.44,A -85,B 0,C 180,E1 3264.189,E2 3264.189} C_VEL
LIN {X 0,Y 554.139,Z 843.44,A -85,B 0,C 180,E1 3269.456,E2 3269.456} C_VEL
LIN {X 0,Y 554.29,Z 843.44,A -85,B 0,C 180,E1 3274.999,E2 3274.999} C_VEL
LIN {X 0,Y 554.079,Z 843.44,A -85,B 0,C 180,E1 3280.977,E2 3280.977} C_VEL
LIN {X 0,Y 554.076,Z 843.44,A -85,B 0,C 180,E1 3287.538,E2 3287.538} C_VEL
LIN {X 0,Y 554.247,Z 843.44,A -85,B 0,C 180,E1 3293.057,E2 3293.057} C_VEL
LIN {X 0,Y 554.402,Z 843.44,A -85,B 0,C 180,E1 3297.266,E2 3297.266} C_VEL
LIN {X 0,Y 562.443,Z 862.278,A -85,B 0,C 180,E1 3298.077,E2 3298.077} C_VEL
LIN {X 0,Y 562.435,Z 913.883,A -85,B 0,C 180,E1 3299.016,E2 3299.016} C_VEL
LIN {X 0,Y 561.428,Z 952.785,A -85,B 0,C 180,E1 3300.332,E2 3300.332} C_VEL
LIN {X 0,Y 560.092,Z 989.507,A -85,B 0,C 180,E1 3302.206,E2 3302.206} C_VEL
LIN {X 0,Y 558.592,Z 1023.908,A -85,B 0,C 180,E1 3304.623,E2 3304.623} C_VEL
LIN {X 0,Y 557.128,Z 1056.13,A -85,B 0,C 180,E1 3307.636,E2 3307.636} C_VEL
LIN {X 0,Y 556.093,Z 1083.044,A -85,B 0,C 180,E1 3310.928,E2 3310.928} C_VEL
LIN {X 0,Y 555.368,Z 1105.035,A -85,B 0,C 180,E1 3314.441,E2 3314.441} C_VEL
LIN {X 0,Y 554.913,Z 1122.496,A -85,B 0,C 180,E1 3318.191,E2 3318.191} C_VEL
LIN {X 0,Y 554.82,Z 1134.258,A -85,B 0,C 180,E1 3321.762,E2 3321.762} C_VEL
LIN {X 0,Y 554.685,Z 1141.501,A -85,B 0,C 180,E1 3325.302,E2 3325.302} C_VEL
LIN {X 0,Y 554.652,Z 1144.612,A -85,B 0,C 180,E1 3328.435,E2 3328.435} C_VEL
LIN {X 0,Y 554.767,Z 1144.554,A -85,B 0,C 180,E1 3331.563,E2 3331.563} C_VEL
LIN {X 0,Y 554.786,Z 1140.044,A -85,B 0,C 180,E1 3335.534,E2 3335.534} C_VEL
LIN {X 0,Y 554.886,Z 1130.581,A -85,B 0,C 180,E1 3339.422,E2 3339.422} C_VEL
LIN {X 0,Y 555.172,Z 1115.388,A -85,B 0,C 180,E1 3343.404,E2 3343.404} C_VEL
LIN {X 0,Y 555.715,Z 1094.796,A -85,B 0,C 180,E1 3347.235,E2 3347.235} C_VEL
LIN {X 0,Y 556.684,Z 1068.119,A -85,B 0,C 180,E1 3350.915,E2 3350.915} C_VEL
LIN {X 0,Y 557.926,Z 1038.546,A -85,B 0,C 180,E1 3354.021,E2 3354.021} C_VEL
LIN {X 0,Y 559.381,Z 1005.957,A -85,B 0,C 180,E1 3356.636,E2 3356.636} C_VEL
LIN {X 0,Y 560.741,Z 972.18,A -85,B 0,C 180,E1 3358.672,E2 3358.672} C_VEL
LIN {X 0,Y 561.934,Z 934.887,A -85,B 0,C 180,E1 3360.265,E2 3360.265} C_VEL
LIN {X 0,Y 562.773,Z 896.053,A -85,B 0,C 180,E1 3361.286,E2 3361.286} C_VEL
LIN {X 0,Y 562.248,Z 861.795,A -85,B 0,C 180,E1 3361.853,E2 3361.853} C_VEL
LIN {X 0,Y 554.109,Z 843.44,A -85,B 0,C 180,E1 3362.659,E2 3362.659} C_VEL
LIN {X 0,Y 554.183,Z 843.44,A -85,B 0,C 180,E1 3368.932,E2 3368.932} C_VEL
LIN {X 0,Y 554.158,Z 843.44,A -85,B 0,C 180,E1 3375.267,E2 3375.267} C_VEL
LIN {X 0,Y 554.105,Z 843.44,A -85,B 0,C 180,E1 3381.068,E2 3381.068} C_VEL
LIN {X 0,Y 554.06,Z 843.44,A -85,B 0,C 180,E1 3386.874,E2 3386.874} C_VEL
LIN {X 0,Y 554.196,Z 843.44,A -85,B 0,C 180,E1 3392.329,E2 3392.329} C_VEL
LIN {X 0,Y 554.301,Z 843.44,A -85,B 0,C 180,E1 3398.238,E2 3398.238} C_VEL
LIN {X 0,Y 554.424,Z 843.44,A -85,B 0,C 180,E1 3404.154,E2 3404.154} C_VEL
LIN {X 0,Y 554.401,Z 843.44,A -85,B 0,C 180,E1 3409.479,E2 3409.479} C_VEL
LIN {X 0,Y 554.531,Z 843.44,A -85,B 0,C 180,E1 3415.303,E2 3415.303} C_VEL
LIN {X 0,Y 554.715,Z 843.44,A -85,B 0,C 180,E1 3421.565,E2 3421.565} C_VEL
LIN {X 0,Y 554.633,Z 843.44,A -85,B 0,C 180,E1 3426.269,E2 3426.269} C_VEL
LIN {X 0,Y 554.334,Z 843.44,A -85,B 0,C 180,E1 3432.621,E2 3432.621} C_VEL
LIN {X 0,Y 554.245,Z 843.44,A -85,B 0,C 180,E1 3437.962,E2 3437.962} C_VEL
LIN {X 0,Y 550.33,Z 843.44,A -85,B 0,C 180,E1 3439.727,E2 3439.727} C_VEL
LIN {X 0,Y 546.352,Z 843.44,A -85,B 0,C 180,E1 3441.518,E2 3441.518} C_VEL
LIN {X 0,Y 546.32,Z 843.44,A -85,B 0,C 180,E1 3447.517,E2 3447.517} C_VEL
LIN {X 0,Y 546.131,Z 843.44,A -85,B 0,C 180,E1 3453.723,E2 3453.723} C_VEL
LIN {X 0,Y 546.206,Z 843.44,A -85,B 0,C 180,E1 3459.607,E2 3459.607} C_VEL
LIN {X 0,Y 546.206,Z 843.44,A -85,B 0,C 180,E1 3463.885,E2 3463.885} C_VEL
LIN {X 0,Y 546.142,Z 843.44,A -85,B 0,C 180,E1 3470.384,E2 3470.384} C_VEL
LIN {X 0,Y 546.165,Z 843.44,A -85,B 0,C 180,E1 3471.872,E2 3471.872} C_VEL
LIN {X 0,Y 555.355,Z 862.547,A -85,B 0,C 180,E1 3472.932,E2 3472.932} C_VEL
LIN {X 0,Y 558.888,Z 871.072,A -85,B 0,C 180,E1 3473.339,E2 3473.339} C_VEL
LIN {X 0,Y 558.124,Z 914.984,A -85,B 0,C 180,E1 3474.205,E2 3474.205} C_VEL
LIN {X 0,Y 556.705,Z 956.21,A -85,B 0,C 180,E1 3475.643,E2 3475.643} C_VEL
LIN {X 0,Y 554.897,Z 994.914,A -85,B 0,C 180,E1 3477.64,E2 3477.64} C_VEL
LIN {X 0,Y 552.801,Z 1032.151,A -85,B 0,C 180,E1 3480.245,E2 3480.245} C_VEL
LIN {X 0,Y 550.768,Z 1067.07,A -85,B 0,C 180,E1 3483.445,E2 3483.445} C_VEL
LIN {X 0,Y 549.135,Z 1097.789,A -85,B 0,C 180,E1 3487.079,E2 3487.079} C_VEL
LIN {X 0,Y 547.927,Z 1123.797,A -85,B 0,C 180,E1 3491.053,E2 3491.053} C_VEL
LIN {X 0,Y 547.314,Z 1142.492,A -85,B 0,C 180,E1 3494.764,E2 3494.764} C_VEL
LIN {X 0,Y 546.961,Z 1157.776,A -85,B 0,C 180,E1 3498.827,E2 3498.827} C_VEL
LIN {X 0,Y 546.829,Z 1167.918,A -85,B 0,C 180,E1 3502.843,E2 3502.843} C_VEL
LIN {X 0,Y 546.751,Z 1173.628,A -85,B 0,C 180,E1 3506.826,E2 3506.826} C_VEL
LIN {X 0,Y 546.742,Z 1175,A -85,B 0,C 180,E1 3510.001,E2 3510.001} C_VEL
LIN {X 0,Y 546.789,Z 1172.094,A -85,B 0,C 180,E1 3514.603,E2 3514.603} C_VEL
LIN {X 0,Y 546.897,Z 1164.401,A -85,B 0,C 180,E1 3518.759,E2 3518.759} C_VEL
LIN {X 0,Y 547.056,Z 1152.3,A -85,B 0,C 180,E1 3522.793,E2 3522.793} C_VEL
LIN {X 0,Y 547.59,Z 1134.045,A -85,B 0,C 180,E1 3527.043,E2 3527.043} C_VEL
LIN {X 0,Y 548.597,Z 1109.777,A -85,B 0,C 180,E1 3531.223,E2 3531.223} C_VEL
LIN {X 0,Y 550.101,Z 1080.266,A -85,B 0,C 180,E1 3535.111,E2 3535.111} C_VEL
LIN {X 0,Y 552.009,Z 1045.418,A -85,B 0,C 180,E1 3538.64,E2 3538.64} C_VEL
LIN {X 0,Y 554.115,Z 1007.893,A -85,B 0,C 180,E1 3541.54,E2 3541.54} C_VEL
LIN {X 0,Y 556.162,Z 967.014,A -85,B 0,C 180,E1 3543.87,E2 3543.87} C_VEL
LIN {X 0,Y 557.81,Z 923.928,A -85,B 0,C 180,E1 3545.546,E2 3545.546} C_VEL
LIN {X 0,Y 559.005,Z 880.201,A -85,B 0,C 180,E1 3546.509,E2 3546.509} C_VEL
LIN {X 0,Y 558.172,Z 867.296,A -85,B 0,C 180,E1 3546.775,E2 3546.775} C_VEL
LIN {X 0,Y 546.389,Z 844.294,A -85,B 0,C 180,E1 3548.08,E2 3548.08} C_VEL
LIN {X 0,Y 546.279,Z 843.44,A -85,B 0,C 180,E1 3548.728,E2 3548.728} C_VEL
LIN {X 0,Y 546.026,Z 843.44,A -85,B 0,C 180,E1 3553.889,E2 3553.889} C_VEL
LIN {X 0,Y 546.222,Z 843.44,A -85,B 0,C 180,E1 3560.395,E2 3560.395} C_VEL
LIN {X 0,Y 546.333,Z 843.44,A -85,B 0,C 180,E1 3566.342,E2 3566.342} C_VEL
LIN {X 0,Y 546.339,Z 843.44,A -85,B 0,C 180,E1 3572.482,E2 3572.482} C_VEL
LIN {X 0,Y 546.216,Z 843.44,A -85,B 0,C 180,E1 3577.167,E2 3577.167} C_VEL
LIN {X 0,Y 546.03,Z 843.44,A -85,B 0,C 180,E1 3580.566,E2 3580.566} C_VEL
LIN {X 0,Y 550.275,Z 861.959,A -85,B 0,C 180,E1 3580.991,E2 3580.991} C_VEL
LIN {X 0,Y 549.959,Z 894.644,A -85,B 0,C 180,E1 3581.667,E2 3581.667} C_VEL
LIN {X 0,Y 549.339,Z 924.044,A -85,B 0,C 180,E1 3582.869,E2 3582.869} C_VEL
LIN {X 0,Y 548.578,Z 952.196,A -85,B 0,C 180,E1 3584.709,E2 3584.709} C_VEL
LIN {X 0,Y 547.844,Z 976.597,A -85,B 0,C 180,E1 3587.024,E2 3587.024} C_VEL
LIN {X 0,Y 547.365,Z 996.373,A -85,B 0,C 180,E1 3589.725,E2 3589.725} C_VEL
LIN {X 0,Y 547.091,Z 1011.716,A -85,B 0,C 180,E1 3592.846,E2 3592.846} C_VEL
LIN {X 0,Y 546.986,Z 1021.029,A -85,B 0,C 180,E1 3596.032,E2 3596.032} C_VEL
LIN {X 0,Y 546.887,Z 1024.389,A -85,B 0,C 180,E1 3598.413,E2 3598.413} C_VEL
LIN {X 0,Y 546.882,Z 1024.311,A -85,B 0,C 180,E1 3601.586,E2 3601.586} C_VEL
LIN {X 0,Y 546.983,Z 1019.028,A -85,B 0,C 180,E1 3604.762,E2 3604.762} C_VEL
LIN {X 0,Y 547.124,Z 1008.033,A -85,B 0,C 180,E1 3607.952,E2 3607.952} C_VEL
LIN {X 0,Y 547.452,Z 993.023,A -85,B 0,C 180,E1 3610.718,E2 3610.718} C_VEL
LIN {X 0,Y 547.971,Z 972.13,A -85,B 0,C 180,E1 3613.378,E2 3613.378} C_VEL
LIN {X 0,Y 548.784,Z 946.178,A -85,B 0,C 180,E1 3615.664,E2 3615.664} C_VEL
LIN {X 0,Y 549.583,Z 917.116,A -85,B 0,C 180,E1 3617.38,E2 3617.38} C_VEL
LIN {X 0,Y 550.098,Z 885.813,A -85,B 0,C 180,E1 3618.491,E2 3618.491} C_VEL
LIN {X 0,Y 549.373,Z 854.365,A -85,B 0,C 180,E1 3619.054,E2 3619.054} C_VEL
LIN {X 0,Y 546.31,Z 843.44,A -85,B 0,C 180,E1 3619.341,E2 3619.341} C_VEL
LIN {X 0,Y 546.287,Z 843.44,A -85,B 0,C 180,E1 3624.563,E2 3624.563} C_VEL
LIN {X 0,Y 546.182,Z 843.44,A -85,B 0,C 180,E1 3630.751,E2 3630.751} C_VEL
LIN {X 0,Y 546.242,Z 843.44,A -85,B 0,C 180,E1 3636.499,E2 3636.499} C_VEL
LIN {X 0,Y 546.136,Z 843.44,A -85,B 0,C 180,E1 3641.705,E2 3641.705} C_VEL
LIN {X 0,Y 546.163,Z 843.44,A -85,B 0,C 180,E1 3648.453,E2 3648.453} C_VEL
LIN {X 0,Y 546.374,Z 843.44,A -85,B 0,C 180,E1 3654.411,E2 3654.411} C_VEL
LIN {X 0,Y 546.477,Z 843.66,A -85,B 0,C 180,E1 3656.744,E2 3656.744} C_VEL
LIN {X 0,Y 555.774,Z 864.744,A -85,B 0,C 180,E1 3657.685,E2 3657.685} C_VEL
LIN {X 0,Y 555.662,Z 913.746,A -85,B 0,C 180,E1 3658.593,E2 3658.593} C_VEL
LIN {X 0,Y 554.532,Z 952.138,A -85,B 0,C 180,E1 3659.896,E2 3659.896} C_VEL
LIN {X 0,Y 553.028,Z 988.222,A -85,B 0,C 180,E1 3661.736,E2 3661.736} C_VEL
LIN {X 0,Y 551.224,Z 1024.082,A -85,B 0,C 180,E1 3664.275,E2 3664.275} C_VEL
LIN {X 0,Y 549.625,Z 1056.123,A -85,B 0,C 180,E1 3667.313,E2 3667.313} C_VEL
LIN {X 0,Y 548.388,Z 1083.04,A -85,B 0,C 180,E1 3670.65,E2 3670.65} C_VEL
LIN {X 0,Y 547.56,Z 1105.805,A -85,B 0,C 180,E1 3674.359,E2 3674.359} C_VEL
LIN {X 0,Y 547.043,Z 1122.494,A -85,B 0,C 180,E1 3678.018,E2 3678.018} C_VEL
LIN {X 0,Y 546.949,Z 1134.257,A -85,B 0,C 180,E1 3681.642,E2 3681.642} C_VEL
LIN {X 0,Y 546.783,Z 1141.732,A -85,B 0,C 180,E1 3685.387,E2 3685.387} C_VEL
LIN {X 0,Y 546.75,Z 1144.612,A -85,B 0,C 180,E1 3688.412,E2 3688.412} C_VEL
LIN {X 0,Y 546.862,Z 1144.554,A -85,B 0,C 180,E1 3691.586,E2 3691.586} C_VEL
LIN {X 0,Y 546.907,Z 1140.281,A -85,B 0,C 180,E1 3695.48,E2 3695.48} C_VEL
LIN {X 0,Y 547.019,Z 1130.583,A -85,B 0,C 180,E1 3699.559,E2 3699.559} C_VEL
LIN {X 0,Y 547.346,Z 1115.392,A -85,B 0,C 180,E1 3703.599,E2 3703.599} C_VEL
LIN {X 0,Y 547.958,Z 1094.857,A -85,B 0,C 180,E1 3707.478,E2 3707.478} C_VEL
LIN {X 0,Y 549.104,Z 1068.124,A -85,B 0,C 180,E1 3711.217,E2 3711.217} C_VEL
LIN {X 0,Y 550.536,Z 1038.555,A -85,B 0,C 180,E1 3714.364,E2 3714.364} C_VEL
LIN {X 0,Y 552.135,Z 1006.01,A -85,B 0,C 180,E1 3717.01,E2 3717.01} C_VEL
LIN {X 0,Y 553.705,Z 971.807,A -85,B 0,C 180,E1 3719.091,E2 3719.091} C_VEL
LIN {X 0,Y 555.121,Z 933.885,A -85,B 0,C 180,E1 3720.712,E2 3720.712} C_VEL
LIN {X 0,Y 556.056,Z 895.044,A -85,B 0,C 180,E1 3721.726,E2 3721.726} C_VEL
LIN {X 0,Y 555.481,Z 864.303,A -85,B 0,C 180,E1 3722.251,E2 3722.251} C_VEL
LIN {X 0,Y 546.166,Z 843.44,A -85,B 0,C 180,E1 3723.271,E2 3723.271} C_VEL
LIN {X 0,Y 546.261,Z 843.44,A -85,B 0,C 180,E1 3729.105,E2 3729.105} C_VEL
LIN {X 0,Y 546.165,Z 843.44,A -85,B 0,C 180,E1 3733.888,E2 3733.888} C_VEL
LIN {X 0,Y 546.19,Z 843.44,A -85,B 0,C 180,E1 3738.458,E2 3738.458} C_VEL
LIN {X 0,Y 546.113,Z 843.44,A -85,B 0,C 180,E1 3744.398,E2 3744.398} C_VEL
LIN {X 0,Y 546.199,Z 843.44,A -85,B 0,C 180,E1 3750.072,E2 3750.072} C_VEL
LIN {X 0,Y 546.356,Z 843.44,A -85,B 0,C 180,E1 3756.138,E2 3756.138} C_VEL
LIN {X 0,Y 546.474,Z 843.44,A -85,B 0,C 180,E1 3760.584,E2 3760.584} C_VEL
LIN {X 0,Y 546.66,Z 843.44,A -85,B 0,C 180,E1 3765.793,E2 3765.793} C_VEL
LIN {X 0,Y 546.583,Z 843.44,A -85,B 0,C 180,E1 3772.04,E2 3772.04} C_VEL
LIN {X 0,Y 546.709,Z 843.44,A -85,B 0,C 180,E1 3776.826,E2 3776.826} C_VEL
LIN {X 0,Y 546.805,Z 843.44,A -85,B 0,C 180,E1 3781.587,E2 3781.587} C_VEL
LIN {X 0,Y 546.725,Z 843.44,A -85,B 0,C 180,E1 3786.36,E2 3786.36} C_VEL
LIN {X 0,Y 546.415,Z 843.44,A -85,B 0,C 180,E1 3792.807,E2 3792.807} C_VEL
LIN {X 0,Y 546.337,Z 843.44,A -85,B 0,C 180,E1 3797.952,E2 3797.952} C_VEL
LIN {X 0,Y 546.352,Z 843.44,A -85,B 0,C 180,E1 3801.518,E2 3801.518} C_VEL
LIN {X 0,Y 542.358,Z 843.44,A -85,B 0,C 180,E1 3803.307,E2 3803.307} C_VEL
LIN {X 0,Y 538.42,Z 843.44,A -85,B 0,C 180,E1 3805.122,E2 3805.122} C_VEL
LIN {X 0,Y 538.279,Z 843.44,A -85,B 0,C 180,E1 3810.416,E2 3810.416} C_VEL
LIN {X 0,Y 538.248,Z 843.44,A -85,B 0,C 180,E1 3816.206,E2 3816.206} C_VEL
LIN {X 0,Y 538.208,Z 843.44,A -85,B 0,C 180,E1 3822.463,E2 3822.463} C_VEL
LIN {X 0,Y 538.161,Z 843.44,A -85,B 0,C 180,E1 3827.528,E2 3827.528} C_VEL
LIN {X 0,Y 538.3,Z 843.989,A -85,B 0,C 180,E1 3831.237,E2 3831.237} C_VEL
LIN {X 0,Y 552.542,Z 872.171,A -85,B 0,C 180,E1 3832.865,E2 3832.865} C_VEL
LIN {X 0,Y 551.66,Z 915.414,A -85,B 0,C 180,E1 3833.733,E2 3833.733} C_VEL
LIN {X 0,Y 550.175,Z 955.384,A -85,B 0,C 180,E1 3835.136,E2 3835.136} C_VEL
LIN {X 0,Y 548.094,Z 993.912,A -85,B 0,C 180,E1 3837.126,E2 3837.126} C_VEL
LIN {X 0,Y 545.749,Z 1031.19,A -85,B 0,C 180,E1 3839.741,E2 3839.741} C_VEL
LIN {X 0,Y 543.544,Z 1065.335,A -85,B 0,C 180,E1 3842.878,E2 3842.878} C_VEL
LIN {X 0,Y 541.778,Z 1094.579,A -85,B 0,C 180,E1 3846.313,E2 3846.313} C_VEL
LIN {X 0,Y 540.387,Z 1120.222,A -85,B 0,C 180,E1 3850.151,E2 3850.151} C_VEL
LIN {X 0,Y 539.603,Z 1140.719,A -85,B 0,C 180,E1 3854.123,E2 3854.123} C_VEL
LIN {X 0,Y 539.096,Z 1157.775,A -85,B 0,C 180,E1 3858.662,E2 3858.662} C_VEL
LIN {X 0,Y 538.946,Z 1167.918,A -85,B 0,C 180,E1 3862.738,E2 3862.738} C_VEL
LIN {X 0,Y 538.87,Z 1173.628,A -85,B 0,C 180,E1 3866.779,E2 3866.779} C_VEL
LIN {X 0,Y 538.853,Z 1175,A -85,B 0,C 180,E1 3870.001,E2 3870.001} C_VEL
LIN {X 0,Y 538.882,Z 1173.627,A -85,B 0,C 180,E1 3873.222,E2 3873.222} C_VEL
LIN {X 0,Y 539.041,Z 1167.915,A -85,B 0,C 180,E1 3877.262,E2 3877.262} C_VEL
LIN {X 0,Y 539.117,Z 1157.771,A -85,B 0,C 180,E1 3881.339,E2 3881.339} C_VEL
LIN {X 0,Y 539.576,Z 1140.71,A -85,B 0,C 180,E1 3885.879,E2 3885.879} C_VEL
LIN {X 0,Y 540.516,Z 1117.959,A -85,B 0,C 180,E1 3890.239,E2 3890.239} C_VEL
LIN {X 0,Y 542.069,Z 1089.662,A -85,B 0,C 180,E1 3894.332,E2 3894.332} C_VEL
LIN {X 0,Y 544.049,Z 1058.137,A -85,B 0,C 180,E1 3897.859,E2 3897.859} C_VEL
LIN {X 0,Y 546.451,Z 1021.059,A -85,B 0,C 180,E1 3901.046,E2 3901.046} C_VEL
LIN {X 0,Y 548.745,Z 982.153,A -85,B 0,C 180,E1 3903.557,E2 3903.557} C_VEL
LIN {X 0,Y 550.857,Z 940.594,A -85,B 0,C 180,E1 3905.456,E2 3905.456} C_VEL
LIN {X 0,Y 552.193,Z 902.229,A -85,B 0,C 180,E1 3906.582,E2 3906.582} C_VEL
LIN {X 0,Y 551.954,Z 870.512,A -85,B 0,C 180,E1 3907.208,E2 3907.208} C_VEL
LIN {X 0,Y 538.553,Z 844.954,A -85,B 0,C 180,E1 3908.725,E2 3908.725} C_VEL
LIN {X 0,Y 538.375,Z 843.44,A -85,B 0,C 180,E1 3908.812,E2 3908.812} C_VEL
LIN {X 0,Y 538.031,Z 843.44,A -85,B 0,C 180,E1 3915.293,E2 3915.293} C_VEL
LIN {X 0,Y 538.339,Z 843.44,A -85,B 0,C 180,E1 3921.778,E2 3921.778} C_VEL
LIN {X 0,Y 538.355,Z 843.44,A -85,B 0,C 180,E1 3927.702,E2 3927.702} C_VEL
LIN {X 0,Y 538.366,Z 843.44,A -85,B 0,C 180,E1 3933.26,E2 3933.26} C_VEL
LIN {X 0,Y 538.252,Z 843.44,A -85,B 0,C 180,E1 3938.552,E2 3938.552} C_VEL
LIN {X 0,Y 538.157,Z 843.652,A -85,B 0,C 180,E1 3940.293,E2 3940.293} C_VEL
LIN {X 0,Y 542.82,Z 864.707,A -85,B 0,C 180,E1 3940.758,E2 3940.758} C_VEL
LIN {X 0,Y 542.384,Z 897.242,A -85,B 0,C 180,E1 3941.487,E2 3941.487} C_VEL
LIN {X 0,Y 541.721,Z 925.917,A -85,B 0,C 180,E1 3942.726,E2 3942.726} C_VEL
LIN {X 0,Y 540.85,Z 953.394,A -85,B 0,C 180,E1 3944.585,E2 3944.585} C_VEL
LIN {X 0,Y 540.067,Z 976.595,A -85,B 0,C 180,E1 3946.834,E2 3946.834} C_VEL
LIN {X 0,Y 539.506,Z 997.244,A -85,B 0,C 180,E1 3949.72,E2 3949.72} C_VEL
LIN {X 0,Y 539.233,Z 1011.713,A -85,B 0,C 180,E1 3952.741,E2 3952.741} C_VEL
LIN {X 0,Y 539.091,Z 1020.041,A -85,B 0,C 180,E1 3955.507,E2 3955.507} C_VEL
LIN {X 0,Y 539.001,Z 1024.387,A -85,B 0,C 180,E1 3958.39,E2 3958.39} C_VEL
LIN {X 0,Y 538.997,Z 1024.31,A -85,B 0,C 180,E1 3961.609,E2 3961.609} C_VEL
LIN {X 0,Y 539.084,Z 1019.031,A -85,B 0,C 180,E1 3964.832,E2 3964.832} C_VEL
